(* CoDeSys 2.3 library: TcNci.lib *)
(* Libraries: TcSystem.lib*27.2.12 14:08:36, TcBaseMath.lib 27.7.04 11:07:56, TcMath.lib 23.9.04 14:15:30, tcnc.lib 10.10.08 16:55:34, standard.lib 5.6.98 11:03:02, TcBase.lib 14.5.09 11:14:08 *)

(* Global variable list: Globale_Variablen *)
VAR_GLOBAL CONSTANT

	NCI_MAX_TOOLDESC:					UDINT := 255; (* in older versions the max number of tool descriptions *)
                                               (* was restricted to 50, cf. issue 1721 & 2365*)

	NCI_MAX_READPREVIEWTABLINES	 	: UINT := 11;
	NCI_MAX_PREVIEWTABLINES 				: UINT := 20;


	(* additional TcNciItp.lib errors *)
	ErrTcNciItp_MFuncReq:			UDINT := 16#4B10;	(* m function request is missing *)
	ErrTcNciItp_ZeroShiftNo:		UDINT	:= 16#4B11;	(* zero shift number is out of range *)
	ErrTcNciItp_RParamIndex:		UDINT	:= 16#4B12;	(* index of r param or size is invalid *)
	ErrTcNciItp_DNo:					UDINT	:= 16#4B13; (* index of d number is out of range *)
	ErrTcNciItp_ItfVersion:			UDINT	:= 16#4B14; (* the cyclic channel interface does not match to the requested function/fb *)
	ErrTcNciItp_NotReady:			UDINT	:= 16#4B15;	(* not ready to support requested function *)
	ErrTcNciItp_NotEnabled:			UDINT	:= 16#4B16;	(* requested function is not enabled *)

	(* states of the interpreter *)
	NCI_INTERPRETER_INITFAILED:	UDINT	:=	0;
	NCI_INTERPRETER_IDLE:			UDINT	:=	1;
	NCI_INTERPRETER_READY:			UDINT	:=	2;
	NCI_INTERPRETER_STARTED:		UDINT	:=	3;
	NCI_INTERPRETER_SCANNING:		UDINT	:=	4;
	NCI_INTERPRETER_RUNNING:		UDINT	:=	5;
	NCI_INTERPRETER_STAY_RUNNING:	UDINT	:=	6;
	NCI_INTERPRETER_WRITETABLE:	UDINT	:=	7;
	NCI_INTERPRETER_SEARCHLINE:	UDINT	:=	8;
	NCI_INTERPRETER_END:				UDINT	:=	9;
	NCI_INTERPRETER_SINGLESTOP:	UDINT	:=	10;
	NCI_INTERPRETER_ABORTING:		UDINT	:=	11;
	NCI_INTERPRETER_ABORTED:		UDINT	:=	12;
	NCI_INTERPRETER_FAULT:			UDINT	:=	13;
	NCI_INTERPRETER_RESET:			UDINT	:=	14;
	NCI_INTERPRETER_STOP:			UDINT := 15;
	NCI_INTERPRETER_WAITFUNC:		UDINT	:=	16;
	NCI_INTERPRETER_FLUSHBUFFERS:	UDINT	:=	17;


END_VAR

VAR_GLOBAL
	g_NcPortTcNci:	UINT	:= AMSPORT_R0_NC;
END_VAR

(* Data type *)
TYPE _ST_ItpInternalPreViewTab :
STRUCT
	nDcTime 		: UDINT := 0;(* T_DCTIME32, timestamp in [ns]) from the NC-SAF(IO)-cycle related to the returned data *)
	nReserved 	: UDINT := 0;(* fill bytes (8 byte alignment) *)
	arrLines		: ARRAY[1..NCI_MAX_READPREVIEWTABLINES] OF ST_ItpPreViewTabLine;(* 272 bytes (8 + 11*24) *)
END_STRUCT
END_TYPE

(* Data type *)
TYPE E_ItpBnMode :
(
	ItpBnm_Abort	:= 0,
	ItpBnm_Adjust	:= 1,
	ItpBnm_Leave	:= 2
);
END_TYPE

(* Data type *)
TYPE E_ItpChannelType :
(
	ItpChannelTypeNone,
	ItpChannelTypeInterpreter,
	ItpChannelTypeKinematic,
	ItpChannelType_InvalidItfVer	:= 16#4B14 (* ErrTcNciItp_ItfVersion  the cyclic channel interface does not match to the requested function/fb *)
);
END_TYPE

(* Data type *)
TYPE E_ItpSingleBlockMode :
(
	ItpSingleBlockOff		:= 0,
	ItpSingleBlockNck		:= 1, (* nc-kernel single block mode *)
	ItpSingleBlockIntp	:= 16#4000 (*interpreter single block mode *)
);
END_TYPE

(* Data type *)
TYPE NciChannelFromPlc :
STRUCT
	nSkipLine		:	WORD;						(* Mask to skip lines *)
	nItpMode		:	WORD;
	nMFuncGranted	:	WORD;						(* granted signal of the M-function *)
	nReserved1		:	ARRAY[7..14] OF BYTE;
	nChaAxesOvr		:	DWORD;					(* Channel override in percent * 10000 *)
	nChaSpindleOvr	:	DWORD;
	nReserved2		:	ARRAY[23..150] OF BYTE;
END_STRUCT
END_TYPE

(* Data type *)
TYPE NciChannelToPlc :
STRUCT
	nJobNo			:	DWORD;
	nFastMFuncMask	:	ARRAY[1..5] OF DWORD;	(* Mask to evaluate fast M-functions *)
	nHskMFuncNo		:	WORD;							(* evaluate M-function with handshake *)
	nHskMFuncReq	: 	WORD;
	nHFuncValue		:	DINT;
	nSpindleRpm		:	WORD;
	nTool				:	WORD;
	nReserved1		:	ARRAY[37..132] OF BYTE; (* 37..40 nChnState *)
                                             (* 41..56 nParams *)
                                             (* 57..88 fParams *)
                                             (* 89..132 reserved *)
	nLoadedProg		:	DWORD;						(* loaded program number if exist *)
	nItpMode			:	WORD;							(* Interpreter mode *)
	nItpState		:	WORD;							(* Interpreter status *)
	nItpErrCode		:	WORD;							(* Interpreter-Channel Error Code *)
	nReserved2		:	ARRAY[143..150] OF BYTE; (*143..144 still reserved *)
                                              (*145..146 nChnId *)
                                              (*147..148 nGrpId *)
                                              (*149..150 nItfVersion *)
END_STRUCT
END_TYPE

(* Data type *)
TYPE ST_ItpEStopParams :
STRUCT
	fDec:		LREAL;
	fJerk:	LREAL;
END_STRUCT
END_TYPE

(* Data type *)
TYPE ST_ItpPreViewTab :
STRUCT
	nDcTime 		: UDINT := 0;(* T_DCTIME32, timestamp in [ns]) from the NC-SAF(IO)-cycle related to the returned data *)
	nReserved 	: UDINT := 0;(* fill bytes (8 byte alignment) *)
	arrLines		: ARRAY[1..NCI_MAX_READPREVIEWTABLINES] OF ST_ItpPreViewTabLine;(* 272 bytes (8 + 11*24) *)
END_STRUCT
END_TYPE

(* Data type *)
TYPE ST_ItpPreViewTabEx :
STRUCT
	nDcTime 		: UDINT := 0;(* T_DCTIME32, timestamp in [ns]) from the NC-SAF(IO)-cycle related to the returned data *)
	nReserved 	: UDINT := 0;(* fill bytes (8 byte alignment) *)
	arrLines		: ARRAY[1..NCI_MAX_PREVIEWTABLINES] OF ST_ItpPreViewTabLine;(* 272 bytes (8 + 11*24) *)
END_STRUCT
END_TYPE

(* Data type *)
TYPE ST_ItpPreViewTabLine :
STRUCT
	fLength 		: LREAL	:= 0.0;
	nBlockNo 	: UDINT 	:= 0;
	nHParam		: UDINT 	:= 0;
	nEntryID		: DINT 	:= 0;
	nReserved	: UDINT 	:= 0;(* fill bytes (8 byte alignment) *)
END_STRUCT
END_TYPE

(* Data type *)
TYPE ST_ItpRetrace :
STRUCT
	nReserved:	ARRAY[1..2] OF DWORD;
	fReserved:	ARRAY[1..8] OF LREAL;
END_STRUCT
END_TYPE

(* Data type *)
TYPE ToolDesc :
STRUCT
	nToolNumber:	UDINT;
	nToolType:		UDINT;
	fParam:			ARRAY[2..15] OF LREAL;
END_STRUCT
END_TYPE

(* Data type *)
TYPE ZeroShiftDesc :
STRUCT
	fShiftX:	LREAL;
	fShiftY:	LREAL;
	fShiftZ:	LREAL;
END_STRUCT
END_TYPE

(* POU MAIN, ST *)
PROGRAM MAIN
VAR
END_VAR
;
END_PROGRAM

(* POU ItpConfirmHsk, ST *)
(* Name:       ItpConfirmHsk                                *)
(* Desc:       confirms the actual m function               *)
(* Author:     kbn                                          *)
(* Date:       30-May-2001                                  *)
(* Revision:   VER 4.0.0                                    *)
(*                                                          *)
(*==========================================================*)

FUNCTION_BLOCK ItpConfirmHsk
VAR_INPUT
	bExecute:	BOOL;
END_VAR
VAR_IN_OUT
	sNciToPlc:	NciChannelToPlc;
	sPlcToNci:	NciChannelFromPlc;
END_VAR
VAR_OUTPUT
	bBusy:	BOOL	:= FALSE;
	bErr:		BOOL	:= FALSE;
	nErrId:	UDINT	:= 0;
END_VAR
VAR
	nState:		UDINT	:= 0;
END_VAR
(*
Version history:
Date          | Version    | created under      | Author          | Remark 
---------------------------------------------------------------------------------------- 
02/01/2002    | 5.1.0      | V2.8.0 (Build 719) | kbn             | modified
              |            |                    |                 | - cycle optimization
---------------------------------------------------------------------------------------- 
*) 
CASE nState OF
0:
	IF bExecute THEN
		bBusy		:= TRUE;
		bErr		:= FALSE;
		nErrId	:= 0;

		IF ItpIsHskMFunc( sNciToPlc ) THEN
			sPlcToNci.nMFuncGranted	:= 1;
			nState	:= 20;
		ELSE
			(* error - there's no request *)
			nState	:= 10;
		END_IF
	END_IF

10:
	(* error in state 0 *)
	(* to ensure a rising edge at bErr we're waiting for the next plc cycle *)
	bErr		:= TRUE;
	nErrId	:= ErrTcNciItp_MFuncReq;
	nState	:= 30;

20:
	(* wait until request bit is gone *)
	(* should be done in the next cycle *)
	IF NOT ItpIsHskMFunc( sNciToPlc ) THEN
		sPlcToNci.nMFuncGranted	:= 0;
		bBusy	:= FALSE;
		IF NOT bExecute THEN
			nState	:= 0;
		ELSE
			(* wait until bExecute has a falling edge *)
			nState	:= 30;
		END_IF
	END_IF

30:
	bBusy	:= FALSE;

	IF NOT bExecute THEN
		nState	:= 0;
	END_IF

END_CASE
END_FUNCTION_BLOCK

(* POU ItpIsHskMFunc, ST *)
(* Name:			ItpIsHskMFunc											*)
(* Desc:			determines if the handshake request bit		*)
(*					is set													*)
(* Author:	 	kbn														*)
(* Date:			30-May-2001												*)
(* Revision:	VER 4.0.0  												*)
(*==========================================================*)

FUNCTION ItpIsHskMFunc : BOOL
VAR_IN_OUT
	sNciToPlc:	NciChannelToPlc;
END_VAR
IF sNciToPlc.nHskMFuncReq <> 0 THEN
	ItpIsHskMFunc	:= TRUE;
ELSE
	ItpIsHskMFunc	:= FALSE;
END_IF
END_FUNCTION

(* POU ItpDelDtg, ST *)
(*==========================================================*)
(* ItpDelDtg																*)
(* Author:	 	kbn														*)
(* Date:			30-May-2001												*)
(* Revision:	VER 5.5.19 												*)
(* last edit:	VER 6.2.33 						                  *)
(*==========================================================*)

FUNCTION_BLOCK ItpDelDtg
VAR_INPUT
	bExecute:	BOOL;
	nChnId:		UDINT;
	tTimeOut:	TIME := DEFAULT_ADS_TIMEOUT;
END_VAR
VAR_OUTPUT
	bBusy:		BOOL	:= FALSE;
	bErr:			BOOL	:= FALSE;
	nErrId:		UDINT	:= 0;
END_VAR
VAR
	nState:		UDINT	:= 0;
	fbAdsWrite:	ADSWRITE;
END_VAR
(*
Version history:
Date          | Version    | created under      | Author          | Remark 
---------------------------------------------------------------------------------------- 
02/01/2002    | 5.1.0      | V2.8.0 (Build 719) | kbn             | modified
              |            |                    |                 | - cycle optimization
---------------------------------------------------------------------------------------- 
06/04/2002    | 5.3.8      | V2.8.0 (Build 733) | kbn             | modified
              |            |                    |                 | - cycle optimization
---------------------------------------------------------------------------------------- 
09/22/2003    | 5.4.13     | V2.9.0 (Build 947) | kbn             | adjustable target port cf. issue #2304
              |            | saved as 2.8       |                 | 
*) 
CASE nState OF

0:
	(* wait on trigger event *)
	IF bExecute THEN
		bBusy	:= TRUE;
		bErr	:= FALSE;
		nErrId	:= 0;

		fbAdsWrite(
			NETID		:= '',
			PORT		:= g_NcPortTcNci,
			IDXGRP	:= NCIDXG_CHN_FUNCS + nChnId,
			IDXOFFS	:= NCIDXO_CHNF_DELDTG,
			LEN		:= 0,
			SRCADDR	:= 0,
			WRITE		:= TRUE,
			TMOUT		:= tTimeOut);

		nState	:= 10;
	END_IF

10:
	(* execute DelDtg command *)
	fbAdsWrite();

	IF NOT fbAdsWrite.BUSY THEN
		IF NOT fbAdsWrite.ERR THEN
			IF NOT bExecute THEN
				fbAdsWrite( WRITE := FALSE );
				nState	:= 0;
			ELSE
				nState	:= 20;
			END_IF
			bBusy	:= FALSE;
		ELSE
			bErr		:= TRUE;
			nErrId	:= fbAdsWrite.ERRID;
			nState	:= 20;
		END_IF
	END_IF
20:
	fbAdsWrite( WRITE := FALSE );
	bBusy	:= FALSE;
	IF NOT bExecute THEN
		nState	:= 0;
	END_IF
END_CASE
END_FUNCTION_BLOCK

(* POU ItpDelDtgEx, ST *)
(*==========================================================*)
(* Name:			ItpDelDtgEx  											*)
(* Desc:			                                             *)
(*             trigger delete distance to go				      *)
(* Author:	 	kbn														*)
(* Date:			26-September-2006										*)
(* last edit:	VER 6.2.33 						                  *)
(*==========================================================*)
FUNCTION_BLOCK ItpDelDtgEx
VAR_IN_OUT
	sNciToPlc:	NciChannelToPlc;
END_VAR
VAR_INPUT
	bExecute:	BOOL;
	tTimeOut:	TIME := DEFAULT_ADS_TIMEOUT;
END_VAR
VAR_OUTPUT
	bBusy:		BOOL	:= FALSE;
	bErr:			BOOL	:= FALSE;
	nErrId:		UDINT	:= 0;
END_VAR
VAR
	nState:			UDINT := 0;
	fbItpDelDtg:	ItpDelDtg;
END_VAR
CASE nState OF
0:
	IF bExecute THEN
		IF ItpGetItfVersion( sNciToPlc ) > 0 THEN
			fbItpDelDtg(
				bExecute	:= TRUE,
				nChnId	:= ItpGetChannelId( sNciToPlc ),
				tTimeOut	:= tTimeOut,
				bBusy	=> bBusy,
				bErr	=> bErr,
				nErrId=> nErrId );
			nState	:= 10;
		ELSE
			bBusy		:= TRUE;
			bErr		:= TRUE;
			nErrId	:= ErrTcNciItp_ItfVersion;
			nState	:= 9999;
		END_IF
	END_IF
10:
	fbItpDelDtg();
	IF NOT fbItpDelDtg.bBusy THEN
		bBusy	:= FALSE;
		IF NOT fbItpDelDtg.bErr THEN
			IF NOT bExecute THEN
				fbItpDelDtg( bExecute := FALSE );
				nState	:= 0;
			ELSE
				nState	:= 9999;
			END_IF
		ELSE
			bErr		:= TRUE;
			nErrId	:= fbItpDelDtg.nErrId;
			nState	:= 9999;
		END_IF
	END_IF

9999:
	fbItpDelDtg( bExecute := FALSE );
	bBusy	:= FALSE;
	IF NOT bExecute THEN
		nState	:= 0;
	END_IF

END_CASE
END_FUNCTION_BLOCK

(* POU ItpGetItfVersion, ST *)
(*==========================================================*)
(* Name:			ItpGetItfVersion										*)
(* Desc:		   determines the interface version of the      *)
(*             cyclic channel interface to plc              *)
(* Author:	 	kbn														*)
(* Date:			26-September-2006										*)
(* last edit:	VER 6.1.21 cf. issue #3209                   *)
(*==========================================================*)
FUNCTION ItpGetItfVersion : UINT
VAR_INPUT
END_VAR
VAR_IN_OUT
	sNciToPlc:	NciChannelToPlc;
END_VAR
VAR
END_VAR
MEMCPY(ADR(ItpGetItfVersion), ADR(sNciToPlc.nReserved2[149]), 2);
END_FUNCTION

(* POU ItpGetChannelId, ST *)
(*==========================================================*)
(* Name:			ItpGetChannelId  										*)
(* Desc:       determines the channel id					      *)
(* Author:	 	kbn														*)
(* Date:			26-September-2006										*)
(* last edit:	VER 6.1.21 cf. issue #3209                   *)
(*==========================================================*)
FUNCTION ItpGetChannelId : UINT
VAR_INPUT
END_VAR
VAR_IN_OUT
	sNciToPlc:	NciChannelToPlc;
END_VAR
VAR
END_VAR
MEMCPY(ADR(ItpGetChannelId), ADR(sNciToPlc.nReserved2[145]), 2);
(*
IF ItpGetItfVersion( sNciToPlc ) > 0 THEN
	MEMCPY(ADR(ItpGetChannelId), ADR(sNciToPlc.nReserved2[145]), 2);
ELSE
	ItpGetChannelId	:= 0;
END_IF
*)
END_FUNCTION

(* POU ItpEnableFeederBackup, ST *)
(*==========================================================*)
(* Name:			ItpEnableFeederBackup    							*)
(* Desc:			THIS IS NOT A RELEASED IMPLEMENTATION AND    *)
(*             SUBJECT TO CHANGE                            *)
(*             enable backup feeder entries for retrace     *)
(* Author:	 	kbn														*)
(* Date:			26-november-2006										*)
(* last edit:	VER 6.2.33 						                  *)
(*==========================================================*)
FUNCTION_BLOCK ItpEnableFeederBackup
VAR_INPUT
	bEnable:		BOOL;
	bExecute:	BOOL;
	tTimeOut:	TIME := DEFAULT_ADS_TIMEOUT;
END_VAR
VAR_IN_OUT
	sNciToPlc:	NciChannelToPlc;
END_VAR
VAR_OUTPUT
	bBusy:		BOOL	:= FALSE;
	bErr:			BOOL	:= FALSE;
	nErrId:		UDINT	:= 0;
END_VAR
VAR
	nState:		UDINT	:= 0;
	nData:		UDINT	:= 0;
	fbAdsWrite:	ADSWRITE;
END_VAR
CASE nState OF
0:
	(* wait on trigger event *)
	IF bExecute THEN
		bBusy	:= TRUE;
		bErr	:= FALSE;
		nErrId	:= 0;

		IF bEnable THEN
			nData	:= 1;
		ELSE
			nData	:= 0;
		END_IF

		fbAdsWrite(
			NETID		:= '',
			PORT		:= g_NcPortTcNci,
			IDXGRP	:= NCIDXG_CHNPARMS + ItpGetChannelId(sNciToPlc:=sNciToPlc),
			IDXOFFS	:= 16#54,
			LEN		:= SIZEOF(nData),
			SRCADDR	:= ADR(nData),
			WRITE		:= TRUE,
			TMOUT		:= tTimeOut);

		nState	:= 10;
	END_IF

10:
	(* execute enable/disable feeder backup*)
	fbAdsWrite();

	IF NOT fbAdsWrite.BUSY THEN
		IF NOT fbAdsWrite.ERR THEN
			IF NOT bExecute THEN
				fbAdsWrite( WRITE := FALSE );
				nState	:= 0;
			ELSE
				nState	:= 20;
			END_IF
			bBusy	:= FALSE;
		ELSE
			bErr		:= TRUE;
			nErrId	:= fbAdsWrite.ERRID;
			nState	:= 20;
		END_IF
	END_IF
20:
	fbAdsWrite( WRITE := FALSE );
	bBusy	:= FALSE;
	IF NOT bExecute THEN
		nState	:= 0;
	END_IF
END_CASE
END_FUNCTION_BLOCK

(* POU ItpEStop, ST *)
(* Name:       ItpEStop                                     *)
(* Desc:       trigger EStop                                *)
(* Author:     kbn                                          *)
(* Date:       29-May-2002                                  *)
(* Revision:   VER 5.4.6                                    *)
(* last edit:	VER 6.2.33 						                  *)
(*==========================================================*)

FUNCTION_BLOCK ItpEStop
VAR_INPUT
	bExecute:	BOOL;
	nGrpId:		UDINT;
	fDec:			LREAL;
	fJerk:		LREAL;
	tTimeOut:	TIME := DEFAULT_ADS_TIMEOUT;
END_VAR
VAR_OUTPUT
	bBusy:	BOOL	:= FALSE;
	bErr:		BOOL	:= FALSE;
	nErrId:	UDINT	:= 0;
END_VAR
VAR
	nState:			UDINT := 0;
	fbAdsWrite:		ADSWRITE;
	stEStopParams:	ST_ItpEStopParams;
END_VAR

(*
Version history:
09/22/2003    | 5.4.13     | V2.9.0 (Build 947) | kbn             | adjustable target port cf. issue #2304
              |            | saved as 2.8       |                 |
*)
CASE nState OF
0:
	IF bExecute THEN
		bBusy		:= TRUE;
		bErr		:= FALSE;
		nErrId	:= 0;

		stEStopParams.fDec	:= fDec;
		stEStopParams.fJerk	:= fJerk;

		fbAdsWrite(
			NETID		:= '',
			PORT		:= AMSPORT_R0_NCSAF,
			IDXGRP	:= 16#3200 + nGrpId,
			IDXOFFS	:= 16#4,
			LEN		:= SIZEOF( stEStopParams ),
			SRCADDR	:= ADR( stEStopParams ),
			WRITE		:= TRUE,
			TMOUT		:= tTimeOut, );

		nState	:= 10;
	END_IF

10:
	fbAdsWrite();

	IF NOT fbAdsWrite.BUSY THEN
		IF NOT fbAdsWrite.ERR THEN
			IF NOT bExecute THEN
				fbAdsWrite( WRITE:= FALSE );
				nState	:= 0;
			ELSE
				nState	:= 20;
			END_IF
			bBusy		:= FALSE;
		ELSE
			bErr		:= TRUE;
			nErrId	:= fbAdsWrite.ERRID;
			nState	:= 20;
		END_IF
	END_IF

20:
	fbAdsWrite( WRITE:= FALSE );
	bBusy		:= FALSE;
	IF NOT bExecute THEN
		nState	:= 0;
	END_IF

END_CASE
END_FUNCTION_BLOCK

(* POU ItpEStopEx, ST *)
(*==========================================================*)
(* Name:			ItpEStopEx  											*)
(* Desc:			triggers E-Stop									   *)
(* Author:	 	kbn														*)
(* Date:			26-September-2006										*)
(* last edit:	VER 6.2.33 						                  *)
(*==========================================================*)

FUNCTION_BLOCK ItpEStopEx
VAR_IN_OUT
	sNciToPlc:	NciChannelToPlc;
END_VAR
VAR_INPUT
	bExecute:	BOOL;
	fDec:			LREAL;
	fJerk:		LREAL;
	tTimeOut:	TIME := DEFAULT_ADS_TIMEOUT;
END_VAR
VAR_OUTPUT
	bBusy:	BOOL	:= FALSE;
	bErr:		BOOL	:= FALSE;
	nErrId:	UDINT	:= 0;
END_VAR
VAR
	nState:			UDINT := 0;
	fbEStop:	ItpEStop;
END_VAR
CASE nState OF
0:
	IF bExecute THEN
		IF ItpGetItfVersion( sNciToPlc ) > 0 THEN
			fbEStop(
				bExecute	:= TRUE,
				nGrpId	:= ItpGetGroupId( sNciToPlc ),
				fDec		:= fDec,
				fJerk		:= fJerk,
				tTimeOut	:= tTimeOut,
				bBusy	=> bBusy,
				bErr	=> bErr,
				nErrId=> nErrId );
			nState	:= 10;
		ELSE
			bBusy		:= TRUE;
			bErr		:= TRUE;
			nErrId	:= ErrTcNciItp_ItfVersion;
			nState	:= 9999;
		END_IF
	END_IF
10:
	fbEStop();
	IF NOT fbEStop.bBusy THEN
		bBusy	:= FALSE;
		IF NOT fbEStop.bErr THEN
			IF NOT bExecute THEN
				fbEStop( bExecute := FALSE );
				nState	:= 0;
			ELSE
				nState	:= 9999;
			END_IF
		ELSE
			bErr		:= TRUE;
			nErrId	:= fbEStop.nErrId;
			nState	:= 9999;
		END_IF
	END_IF

9999:
	fbEStop( bExecute := FALSE );
	bBusy	:= FALSE;
	IF NOT bExecute THEN
		nState	:= 0;
	END_IF

END_CASE
END_FUNCTION_BLOCK

(* POU ItpGetGroupId, ST *)
(*==========================================================*)
(* Name:			ItpGetGroupId 											*)
(* Desc:	      determines the group id						      *)
(* Author:	 	kbn														*)
(* Date:			26-September-2006										*)
(* last edit:	VER 6.1.21 cf. issue #3209                   *)
(*==========================================================*)
FUNCTION ItpGetGroupId : UINT
VAR_INPUT
END_VAR
VAR_IN_OUT
	sNciToPlc:	NciChannelToPlc;
END_VAR
VAR
END_VAR
MEMCPY(ADR(ItpGetGroupId), ADR(sNciToPlc.nReserved2[147]), 2);
(*
IF ItpGetItfVersion( sNciToPlc ) > 0 THEN
	MEMCPY(ADR(ItpGetGroupId), ADR(sNciToPlc.nReserved2[147]), 2);
ELSE
	ItpGetGroupId	:= 0;
END_IF
*)
END_FUNCTION

(* POU ItpGetBlockNumber, ST *)
(* Name:			ItpGetBlockNumber										*)
(* Desc:			Returns the currrent block number				*)
(*						of the NC program									*)
(*	Author:	 	bw															*)
(* Date:			27-Nov-2012												*)
(* Revision:	VER 1.0.0  												*)
(*==========================================================*)
FUNCTION ItpGetBlockNumber : UDINT
VAR_IN_OUT
	sNciToPlc:	NciChannelToPlc;
END_VAR
ItpGetBlockNumber := sNciToPlc.nJobNo;
END_FUNCTION

(* POU ItpGetBottleNeckLookAhead, ST *)
(* Name:			ItpGetBottleNeckLookAhead  						*)
(* Desc:			gets the size of the look ahead for the 		*)
(*             contour collision detection (bottle neck)    *)
(* Author:	 	kbn														*)
(* Date:			26-March-2002											*)
(* Revision:	VER 5.3.4  												*)
(* last edit:	VER 6.2.33 						                  *)
(*==========================================================*)

FUNCTION_BLOCK ItpGetBottleNeckLookAhead
VAR_INPUT
	bExecute:	BOOL;
	nChnId:		UDINT;
	tTimeOut:	TIME := DEFAULT_ADS_TIMEOUT;
END_VAR
VAR_OUTPUT
	bBusy:	BOOL;
	bErr:		BOOL;
	nErrId:	UDINT;
	nLookAhead:	UDINT;
END_VAR
VAR
	nState:		UDINT	:= 0;
	fbAdsRead:	ADSREAD;
END_VAR
VAR CONSTANT
	IDXO_CHNP_BNLOOKAHEAD:	UDINT	:= 16#51;
END_VAR

(*
Version history:
09/22/2003    | 5.4.13     | V2.9.0 (Build 947) | kbn             | adjustable target port cf. issue #2304
              |            | saved as 2.8       |                 |
*)
CASE nState OF

0:
	(* wait on trigger event *)
	IF bExecute THEN
		bBusy		:= TRUE;
		bErr		:= FALSE;
		nErrId	:= 0;

		fbAdsRead(
			NETID		:= '',
			PORT		:= g_NcPortTcNci,
			IDXGRP	:= NCIDXG_CHN_PARMS + nChnId,
			IDXOFFS	:= IDXO_CHNP_BNLOOKAHEAD,
			LEN		:= SIZEOF( nLookAhead ),
			DESTADDR	:= ADR( nLookAhead ),
			READ		:= TRUE,
			TMOUT		:= tTimeOut );

		nState	:= 10;
	END_IF

10:
	fbAdsRead();

	IF NOT fbAdsRead.BUSY THEN
		IF NOT fbAdsRead.ERR THEN
			IF NOT bExecute THEN
				fbAdsRead( READ := FALSE );
				nState	:= 0;
			ELSE
				nState	:= 20;
			END_IF
			bBusy	:= FALSE;
		ELSE
			bErr		:= TRUE;
			nErrId	:= fbAdsRead.ERRID;
			nState	:= 20;
		END_IF
	END_IF

20:
	fbAdsRead( READ := FALSE );
	bBusy	:= FALSE;

	IF NOT bExecute THEN
		nState	:= 0;
	END_IF

END_CASE
END_FUNCTION_BLOCK

(* POU ItpGetBottleNeckLookAheadEx, ST *)
(*==========================================================*)
(* Name:			ItpGetBottleNeckLookAheadEx						*)
(* Desc:			gets the size of the look ahead for the 		*)
(*             contour collision detection (bottle neck)    *)
(* Author:	 	kbn														*)
(* Date:			26-September-2006										*)
(* last edit:	VER 6.2.33 						                  *)
(*==========================================================*)

FUNCTION_BLOCK ItpGetBottleNeckLookAheadEx
VAR_INPUT
	bExecute:	BOOL;
	tTimeOut:	TIME := DEFAULT_ADS_TIMEOUT;
END_VAR
VAR_IN_OUT
	sNciToPlc:	NciChannelToPlc;
END_VAR
VAR_OUTPUT
	bBusy:	BOOL;
	bErr:		BOOL;
	nErrId:	UDINT;
	nLookAhead:	UDINT;
END_VAR
VAR
	nState:		UDINT := 0;
	fbItpGetBottleNeckLookAhead:	ItpGetBottleNeckLookAhead;
END_VAR
CASE nState OF
0:
	IF bExecute THEN
		IF ItpGetItfVersion( sNciToPlc ) > 0 THEN
			fbItpGetBottleNeckLookAhead(
				bExecute	:= TRUE,
				nChnId	:= ItpGetChannelId( sNciToPlc ),
				tTimeOut	:= tTimeOut,
				bBusy	=> bBusy,
				bErr	=> bErr,
				nErrId=> nErrId,
				nLookAhead=>nLookAhead );
			nState	:= 10;
		ELSE
			bBusy		:= TRUE;
			bErr		:= TRUE;
			nErrId	:= ErrTcNciItp_ItfVersion;
			nState	:= 9999;
		END_IF
	END_IF
10:
	fbItpGetBottleNeckLookAhead( nLookAhead=>nLookAhead );
	IF NOT fbItpGetBottleNeckLookAhead.bBusy THEN
		bBusy	:= FALSE;
		IF NOT fbItpGetBottleNeckLookAhead.bErr THEN
			IF NOT bExecute THEN
				fbItpGetBottleNeckLookAhead( bExecute := FALSE, nLookAhead=>nLookAhead );
				nState	:= 0;
			ELSE
				nState	:= 9999;
			END_IF
		ELSE
			bErr		:= TRUE;
			nErrId	:= fbItpGetBottleNeckLookAhead.nErrId;
			nState	:= 9999;
		END_IF
	END_IF

9999:
	fbItpGetBottleNeckLookAhead( bExecute:=FALSE, nLookAhead=>nLookAhead );
	bBusy	:= FALSE;
	IF NOT bExecute THEN
		nState	:= 0;
	END_IF

END_CASE
END_FUNCTION_BLOCK

(* POU ItpGetBottleNeckMode, ST *)
(* Name:			ItpGetBottleNeckMode        						*)
(* Desc:			get the reaction mode for the contour        *)
(*             collision detection                          *)
(* Author:	 	kbn														*)
(* Date:			26-March-2002											*)
(* Revision:	VER 5.3.4  												*)
(* last edit:	VER 6.2.33 						                  *)
(*==========================================================*)

FUNCTION_BLOCK ItpGetBottleNeckMode
VAR_INPUT
	bExecute:			BOOL;
	nChnId:				UDINT;
	tTimeOut:			TIME := DEFAULT_ADS_TIMEOUT;
END_VAR
VAR_OUTPUT
	bBusy:	BOOL;
	bErr:		BOOL;
	nErrId:	UDINT;
	eBottleNeckMode:	E_ItpBnMode;
END_VAR
VAR
	nState:		UDINT	:= 0;
	fbAdsRead:	ADSREAD;
	nTemp:		UDINT;
END_VAR
VAR CONSTANT
	IDXO_CHNP_BNMODE:	UDINT	:= 16#50;
END_VAR

(*
Version history:
09/22/2003    | 5.4.13     | V2.9.0 (Build 947) | kbn             | adjustable target port cf. issue #2304
              |            | saved as 2.8       |                 |
*)
CASE nState OF

0:
	(* wait on trigger event *)
	IF bExecute THEN
		bBusy		:= TRUE;
		bErr		:= FALSE;
		nErrId	:= 0;

		fbAdsRead(
			NETID		:= '',
			PORT		:= g_NcPortTcNci,
			IDXGRP	:= NCIDXG_CHN_PARMS + nChnId,
			IDXOFFS	:= IDXO_CHNP_BNMODE,
			LEN		:= SIZEOF( nTemp ),
			DESTADDR	:= ADR( nTemp ),
			READ		:= TRUE,
			TMOUT		:= tTimeOut );

		nState	:= 10;
	END_IF

10:
	fbAdsRead();

	IF NOT fbAdsRead.BUSY THEN
		IF NOT fbAdsRead.ERR THEN
			eBottleNeckMode	:= UDINT_TO_INT( nTemp );
			IF NOT bExecute THEN
				fbAdsRead( READ := FALSE );
				nState	:= 0;
			ELSE
				nState	:= 20;
			END_IF
			bBusy	:= FALSE;
		ELSE
			bErr		:= TRUE;
			nErrId	:= fbAdsRead.ERRID;
			nState	:= 20;
		END_IF
	END_IF

20:
	fbAdsRead( READ := FALSE );
	bBusy	:= FALSE;

	IF NOT bExecute THEN
		nState	:= 0;
	END_IF

END_CASE
END_FUNCTION_BLOCK

(* POU ItpGetBottleNeckModeEx, ST *)
(*==========================================================*)
(* Name:			ItpGetBottleNeckModeEx								*)
(* Desc:			returns the reaction mode for the contour    *)
(*             collision detection                          *)
(* Author:	 	kbn														*)
(* Date:			26-September-2006										*)
(* last edit:	VER 6.2.33 						                  *)
(*==========================================================*)
FUNCTION_BLOCK ItpGetBottleNeckModeEx
VAR_INPUT
	bExecute:			BOOL;
	tTimeOut:			TIME := DEFAULT_ADS_TIMEOUT;
END_VAR
VAR_IN_OUT
	sNciToPlc:	NciChannelToPlc;
END_VAR
VAR_OUTPUT
	bBusy:	BOOL;
	bErr:		BOOL;
	nErrId:	UDINT;
	eBottleNeckMode:	E_ItpBnMode;
END_VAR
VAR
	nState:		UDINT := 0;
	fbItpGetBottleNeckMode:	ItpGetBottleNeckMode;
END_VAR
CASE nState OF
0:
	IF bExecute THEN
		IF ItpGetItfVersion( sNciToPlc ) > 0 THEN
			fbItpGetBottleNeckMode(
				bExecute	:= TRUE,
				nChnId	:= ItpGetChannelId( sNciToPlc ),
				tTimeOut	:= tTimeOut,
				bBusy	=> bBusy,
				bErr	=> bErr,
				nErrId=> nErrId,
				eBottleNeckMode=> eBottleNeckMode );
			nState	:= 10;
		ELSE
			bBusy		:= TRUE;
			bErr		:= TRUE;
			nErrId	:= ErrTcNciItp_ItfVersion;
			nState	:= 9999;
		END_IF
	END_IF
10:
	fbItpGetBottleNeckMode( eBottleNeckMode=>eBottleNeckMode );
	IF NOT fbItpGetBottleNeckMode.bBusy THEN
		bBusy	:= FALSE;
		IF NOT fbItpGetBottleNeckMode.bErr THEN
			IF NOT bExecute THEN
				fbItpGetBottleNeckMode( bExecute := FALSE, eBottleNeckMode=>eBottleNeckMode );
				nState	:= 0;
			ELSE
				nState	:= 9999;
			END_IF
		ELSE
			bErr		:= TRUE;
			nErrId	:= fbItpGetBottleNeckMode.nErrId;
			nState	:= 9999;
		END_IF
	END_IF

9999:
	fbItpGetBottleNeckMode( bExecute:=FALSE, eBottleNeckMode=>eBottleNeckMode );
	bBusy	:= FALSE;
	IF NOT bExecute THEN
		nState	:= 0;
	END_IF

END_CASE
END_FUNCTION_BLOCK

(* POU ItpGetChannelType, ST *)
(* Name:			ItpGetChannelType										*)
(* Desc:			Returns the Channel type as an Enum				*)
(*	Author:	 	bw															*)
(* Date:			27-Nov-2012												*)
(* Revision:	VER 1.0.0  												*)
(*==========================================================*)
FUNCTION ItpGetChannelType : E_ItpChannelType
VAR_IN_OUT
	sNciToPlc:	NciChannelToPlc;
END_VAR
IF ItpGetItfVersion(sNciToPlc)>=6 THEN
	CASE (sNciToPlc.nReserved1[37] AND 2#00000011) OF
		0:	ItpGetChannelType := ItpChannelTypeNone;
		1:	ItpGetChannelType := ItpChannelTypeInterpreter;
		2:	ItpGetChannelType := ItpChannelTypeKinematic;
		3:	ItpGetChannelType := ItpChannelTypeNone;
		ELSE
			ItpGetChannelType := ItpChannelTypeNone;
	END_CASE
ELSE
	ItpGetChannelType := ItpChannelType_InvalidItfVer;
END_IF
END_FUNCTION

(* POU ItpGetCyclicLRealOffsets, ST *)
(*==========================================================*)
(* Name:			ItpGetCyclicLRealOffsets							*)
(* Desc:			THIS IS NOT A RELEASED IMPLEMENTATION AND    *)
(*             SUBJECT TO CHANGE                            *)
(*             specifies index offsets for cylcic channel   *)
(*             interface                                    *)
(* Author:	 	kbn														*)
(* Date:			08-October-2007										*)
(* last edit:	VER 6.2.33 						                  *)
(*==========================================================*)
FUNCTION_BLOCK ItpGetCyclicLRealOffsets
VAR_INPUT
	bExecute:	BOOL;
	tTimeOut:	TIME := DEFAULT_ADS_TIMEOUT;
END_VAR
VAR_IN_OUT
	sNciToPlc:	NciChannelToPlc;
END_VAR
VAR_OUTPUT
	bBusy:		BOOL	:= FALSE;
	bErr:			BOOL	:= FALSE;
	nErrId:		UDINT	:= 0;
	nIndexOffsetParam1:	UDINT := 0;
	nIndexOffsetParam2:	UDINT := 0;
	nIndexOffsetParam3:	UDINT := 0;
	nIndexOffsetParam4:	UDINT := 0;
END_VAR
VAR
	nState:	UDINT	:= 0;
	nIndexOffsets: ARRAY[1..4] OF UDINT;
	fbAdsRead:		ADSREAD;
END_VAR
CASE nState OF
0:
	IF  bExecute THEN
		bBusy	:= TRUE;
		bErr	:= FALSE;
		nErrId	:= 0;
		fbAdsRead(
			NETID		:= '',
			PORT		:= g_NcPortTcNci,
			IDXGRP	:= NCIDXG_CHNPARMS + ItpGetChannelId(sNciToPlc:=sNciToPlc),
			IDXOFFS	:= 16#56,
			LEN		:= SIZEOF( nIndexOffsets ),
			DESTADDR	:= ADR( nIndexOffsets ),
			READ		:= TRUE,
			TMOUT		:= tTimeOut );
		nState	:= 10;
	END_IF

10:
	fbAdsRead();

	IF NOT fbAdsRead.BUSY THEN
		IF NOT fbAdsRead.ERR THEN

		nIndexOffsetParam1	:= nIndexOffsets[1] ;
		nIndexOffsetParam2	:= nIndexOffsets[2] ;
		nIndexOffsetParam3	:= nIndexOffsets[3] ;
		nIndexOffsetParam4	:= nIndexOffsets[4] ;

			IF NOT bExecute THEN
				fbAdsRead( READ := FALSE );
				nState	:= 0;
			ELSE
				nState	:= 20;
			END_IF
			bBusy		:= FALSE;
		ELSE
			bErr		:= TRUE;
			nErrId	:= fbAdsRead.ERRID;
			nState	:= 20;
		END_IF
	END_IF

20:
	fbAdsRead( READ:= FALSE );
	bBusy		:= FALSE;
	IF NOT bExecute THEN
		nState	:= 0;
	END_IF

END_CASE
END_FUNCTION_BLOCK

(* POU ItpGetCyclicUdintOffsets, ST *)
(*==========================================================*)
(* Name:			ItpGetCyclicUdintOffsets							*)
(* Desc:			THIS IS NOT A RELEASED IMPLEMENTATION AND    *)
(*             SUBJECT TO CHANGE                            *)
(*             specifies index offsets for cylcic channel   *)
(*             interface                                    *)
(* Author:	 	kbn														*)
(* Date:			08-October-2007										*)
(* last edit:	VER 6.2.33 						                  *)
(*==========================================================*)
FUNCTION_BLOCK ItpGetCyclicUdintOffsets
VAR_INPUT
	bExecute:	BOOL;
	tTimeOut:	TIME := DEFAULT_ADS_TIMEOUT;
END_VAR
VAR_IN_OUT
	sNciToPlc:	NciChannelToPlc;
END_VAR
VAR_OUTPUT
	bBusy:		BOOL	:= FALSE;
	bErr:			BOOL	:= FALSE;
	nErrId:		UDINT	:= 0;
	nIndexOffsetParam1:	UDINT := 0;
	nIndexOffsetParam2:	UDINT := 0;
	nIndexOffsetParam3:	UDINT := 0;
	nIndexOffsetParam4:	UDINT := 0;
END_VAR
VAR
	nState:	UDINT	:= 0;
	nIndexOffsets: ARRAY[1..4] OF UDINT;
	fbAdsRead:		ADSREAD;
END_VAR
CASE nState OF
0:
	IF  bExecute THEN
		bBusy	:= TRUE;
		bErr	:= FALSE;
		nErrId	:= 0;
		fbAdsRead(
			NETID		:= '',
			PORT		:= g_NcPortTcNci,
			IDXGRP	:= NCIDXG_CHNPARMS + ItpGetChannelId(sNciToPlc:=sNciToPlc),
			IDXOFFS	:= 16#55,
			LEN		:= SIZEOF( nIndexOffsets ),
			DESTADDR	:= ADR( nIndexOffsets ),
			READ		:= TRUE,
			TMOUT		:= tTimeOut );
		nState	:= 10;
	END_IF

10:
	fbAdsRead();

	IF NOT fbAdsRead.BUSY THEN
		IF NOT fbAdsRead.ERR THEN

		nIndexOffsetParam1	:= nIndexOffsets[1] ;
		nIndexOffsetParam2	:= nIndexOffsets[2] ;
		nIndexOffsetParam3	:= nIndexOffsets[3] ;
		nIndexOffsetParam4	:= nIndexOffsets[4] ;

			IF NOT bExecute THEN
				fbAdsRead( READ := FALSE );
				nState	:= 0;
			ELSE
				nState	:= 20;
			END_IF
			bBusy		:= FALSE;
		ELSE
			bErr		:= TRUE;
			nErrId	:= fbAdsRead.ERRID;
			nState	:= 20;
		END_IF
	END_IF

20:
	fbAdsRead( READ:= FALSE );
	bBusy		:= FALSE;
	IF NOT bExecute THEN
		nState	:= 0;
	END_IF

END_CASE
END_FUNCTION_BLOCK

(* POU ItpGetError, ST *)
(* Name:			ItpGetError												*)
(* Desc:			returns the error number							*)
(* Author:	 	kbn														*)
(* Date:			30-May-2001												*)
(* Revision:	VER 4.0.0  												*)
(*==========================================================*)

FUNCTION ItpGetError : UINT
VAR_IN_OUT
	sNciToPlc:	NciChannelToPlc;
END_VAR
VAR
END_VAR
ItpGetError	:= sNciToPlc.nItpErrCode;
END_FUNCTION

(* POU ItpGetGeoInfoAndHParam, ST *)
FUNCTION_BLOCK ItpGetGeoInfoAndHParam
VAR_IN_OUT
	sNciToPlc:	NciChannelToPlc;
END_VAR
VAR_OUTPUT
	stTab		: ST_ItpPreViewTab;
	nErrId	: UDINT;
END_VAR
{library private}
VAR
	fbCall	: FW_CallGenericFb := ( funGrp := GENERIC_FB_GRP_NC, funNum:= GENERIC_FB_NC_GETGEOINFOANDHPARAM );
	in 		: ARRAY[0..1] OF UDINT;(* 8 byte = nGrpId, nSubIdx *)
END_VAR
IF ItpGetItfVersion( sNciToPlc ) < 5 THEN
	nErrId	:= ErrTcNciItp_ItfVersion;
	RETURN;
END_IF


(* prepare input params *)
in[0] := ItpGetGroupId( sNciToPlc );
in[1] := 0; (* reserved for certain bit mask *)

(* call firmware function block *)
fbCall(	pWrite := ADR( in ), cbWrite:= SIZEOF( in ), pRead := ADR( stTab ), cbRead := SIZEOF( stTab ), nErrID=>nErrID );
END_FUNCTION_BLOCK

(* POU ItpGetGeoInfoAndHParamEx, ST *)
FUNCTION_BLOCK ItpGetGeoInfoAndHParamEx
(* Extended FB for reading geometric information from Nci channel 						*)
(* The H-Parameter Value is based an segment end and 10 past path values are stored		*)
VAR_IN_OUT
	sNciToPlc				: NciChannelToPlc;
END_VAR
VAR_OUTPUT
	stTab					: ST_ItpPreViewTabEx;
	nErrId 					: UDINT;
END_VAR		
{library private}
VAR
	fbCall					: FW_CallGenericFb := ( funGrp := GENERIC_FB_GRP_NC, funNum:= GENERIC_FB_NC_GETGEOINFOANDHPARAM );
	in 						: ARRAY[0..1] OF UDINT;(* 8 byte = nGrpId, nSubIdx *)

	PathInfoOffset				: DINT;
	stReadTab				: ST_ItpPreViewTab;
	stLastReadTab			: ST_ItpPreViewTab;
	stInternalTab				: ST_ItpPreViewTabEx;
	stLastInternalTab			: ST_ItpPreViewTabEx;

	NoOfNewPastEntries		: DINT;
	PathLengthCorrection		: LREAL;

	i,j						: DINT;

	DataError				: BOOL;

	(* Debug *)
	debugcounterZeroData	: UDINT;

	LastPathId				: UDINT;
END_VAR
IF ItpGetItfVersion( sNciToPlc ) < 5 THEN
	nErrId	:= ErrTcNciItp_ItfVersion;
	RETURN;
END_IF

(* prepare input params *)
in[0] := ItpGetGroupId(sNciToPlc);
in[1] := 0; (* reserved for certain bit mask *)

(* call firmware function block *)
fbCall(	pWrite := ADR( in ), cbWrite:= SIZEOF( in ), pRead := ADR( stReadTab ), cbRead := SIZEOF( stReadTab ), nErrID=>nErrId );

IF nErrId <> 0 THEN
	MEMSET(ADR(stReadTab),0,SIZEOF(stReadTab));
	MEMSET(ADR(stLastReadTab),0,SIZEOF(stLastReadTab));
	MEMSET(ADR(stInternalTab),0,SIZEOF(stInternalTab));
	MEMSET(ADR(stLastInternalTab),0,SIZEOF(stLastInternalTab));
	PathLengthCorrection := 0;
	RETURN;
END_IF

(*Init Path Position Info*)
PathInfoOffset := NCI_MAX_PREVIEWTABLINES - NCI_MAX_READPREVIEWTABLINES + 1;

FOR i := 1 TO NCI_MAX_PREVIEWTABLINES DO
	stInternalTab.arrLines[i].nEntryID:=0;
	stInternalTab.arrLines[i].nHParam:=0;
	stInternalTab.arrLines[i].fLength:=0;
	stInternalTab.arrLines[i].nBlockNo:=0;

	stTab:=stInternalTab;
END_FOR

(*Zero data recieved *)
DataError := TRUE;
FOR i := 1 TO NCI_MAX_READPREVIEWTABLINES DO
	IF  (stReadTab.arrLines[i].nEntryID > 0) THEN
		DataError := FALSE;
	END_IF
END_FOR

IF DataError THEN 
	nErrId := 9998;

	MEMSET(ADR(stReadTab),0,SIZEOF(stReadTab));
	MEMSET(ADR(stLastReadTab),0,SIZEOF(stLastReadTab));
	MEMSET(ADR(stInternalTab),0,SIZEOF(stInternalTab));
	MEMSET(ADR(stLastInternalTab),0,SIZEOF(stLastInternalTab));
	PathLengthCorrection := 0;
	debugcounterZeroData := debugcounterZeroData + 1;

	RETURN;
ELSIF nErrId = 0 THEN
	stInternalTab.nDcTime := stReadTab.nDcTime;
	stInternalTab.nReserved := stReadTab.nReserved;

	(* Create new  entries *)
	FOR i := 1 TO NCI_MAX_READPREVIEWTABLINES-1 DO
		IF stReadTab.arrLines[i+1].nEntryID > 0 THEN
			stInternalTab.arrLines[i+PathInfoOffset] := stReadTab.arrLines[i];
			stInternalTab.arrLines[i+PathInfoOffset].nHParam := stReadTab.arrLines[i+1].nHParam;
		END_IF
	END_FOR

	(* Delete buffered entries which have recieved new path lengths and calculate pathlength correction *)
	FOR i := NCI_MAX_PREVIEWTABLINES TO PathInfoOffset+1 BY -1 DO
		FOR j := NCI_MAX_PREVIEWTABLINES TO 1 BY -1 DO
			IF stLastInternalTab.arrLines[j].nEntryID = stInternalTab.arrLines[i].nEntryID THEN
				IF j > PathInfoOffset THEN
					PathLengthCorrection := stLastInternalTab.arrLines[j].fLength - stInternalTab.arrLines[i].fLength;
				END_IF
				stLastInternalTab.arrLines[j].fLength:=0;
				stLastInternalTab.arrLines[j].nEntryID:=0;
				stLastInternalTab.arrLines[j].nHParam:=0;	
			END_IF 
		END_FOR
	END_FOR

	(* Update past entries already buffered *)
	FOR i := PathInfoOffset  TO 1 BY -1 DO
		stInternalTab.arrLines[i] := stLastInternalTab.arrLines[i];
		IF stLastInternalTab.arrLines[i].nEntryID > 0 THEN
			stInternalTab.arrLines[i].fLength := stInternalTab.arrLines[i].fLength - PathLengthCorrection;
		END_IF
	END_FOR

	(*Remove Zero Enties *)
	FOR i := PathInfoOffset  TO 1 BY -1 DO
		IF stInternalTab.arrLines[i].nEntryID = 0 THEN
			IF i > 1 THEN
				FOR j := i  TO 2 BY -1 DO
					stInternalTab.arrLines[j] :=stInternalTab.arrLines[j-1]; 
				END_FOR			
			END_IF
			stLastInternalTab.arrLines[1].fLength:=0;
			stLastInternalTab.arrLines[1].nEntryID:=0;
			stLastInternalTab.arrLines[1].nHParam:=0;	
		END_IF
	END_FOR

	(* Check new past entries *)
	NoOfNewPastEntries := 0;
	FOR i := NCI_MAX_PREVIEWTABLINES TO PathInfoOffset+1 BY -1 DO
		IF stLastInternalTab.arrLines[i].nEntryID > 0 THEN
			NoOfNewPastEntries := NoOfNewPastEntries + 1;
		END_IF
	END_FOR

	(* Add new entries to FIFO, If full oldest entries are deleted *)
	IF NoOfNewPastEntries > 0 THEN
		FOR i := 1 TO (PathInfoOffset - NoOfNewPastEntries)DO
			stInternalTab.arrLines[i] := stInternalTab.arrLines[i+NoOfNewPastEntries];
		END_FOR
		j:=PathInfoOffset+1;
		FOR i := NCI_MAX_PREVIEWTABLINES TO PathInfoOffset+1 BY -1 DO
			IF stLastInternalTab.arrLines[i].nEntryID > 0 THEN
				j:=j-1;
				stInternalTab.arrLines[j] := stLastInternalTab.arrLines[i];
				stInternalTab.arrLines[j].fLength := stInternalTab.arrLines[j].fLength - PathLengthCorrection;
			END_IF
		END_FOR
	END_IF

	stTab := stInternalTab;

	stLastReadTab := stReadTab;
	stLastInternalTab := stTab;

	LastPathId := stTab.arrLines[10].nEntryID;
END_IF
END_FUNCTION_BLOCK

(* POU ItpGetGroupAxisIds, ST *)
(* Name:			ItpGetGroupAxisIds									*)
(* Desc:			Outputs a list of the Group Axes 				*)
(*						or returns an interface version error		*)
(*	Author:	 	bw															*)
(* Date:			02-Feb-2012												*)
(* Revision:	VER 1.0.0  												*)
(*==========================================================*)

FUNCTION ItpGetGroupAxisIds : DWORD
VAR_INPUT
END_VAR
VAR_IN_OUT
	nNciAxisIds 	: 	ARRAY[1..8] OF DWORD;		(*A list of Axes built in the Group*)
	sNciToPlc		:	NciChannelToPlc;
END_VAR
VAR
END_VAR
IF ItpGetItfVersion(sNciToPlc)>=6 THEN
	ItpGetGroupAxisIds	:= 0;
	nNciAxisIds[1] := BYTE_TO_DWORD(sNciToPlc.nReserved1[89]);
	nNciAxisIds[2] := BYTE_TO_DWORD(sNciToPlc.nReserved1[90]);
	nNciAxisIds[3] := BYTE_TO_DWORD(sNciToPlc.nReserved1[91]);
	nNciAxisIds[4] := BYTE_TO_DWORD(sNciToPlc.nReserved1[92]);
	nNciAxisIds[5] := BYTE_TO_DWORD(sNciToPlc.nReserved1[93]);
	nNciAxisIds[6] := BYTE_TO_DWORD(sNciToPlc.nReserved1[94]);
	nNciAxisIds[7] := BYTE_TO_DWORD(sNciToPlc.nReserved1[95]);
	nNciAxisIds[8] := BYTE_TO_DWORD(sNciToPlc.nReserved1[96]);
ELSE
	ItpGetGroupAxisIds := ErrTcNciItp_ItfVersion;
	nNciAxisIds[1] := 0;
	nNciAxisIds[2] := 0;
	nNciAxisIds[3] := 0;
	nNciAxisIds[4] := 0;
	nNciAxisIds[5] := 0;
	nNciAxisIds[6] := 0;
	nNciAxisIds[7] := 0;
	nNciAxisIds[8] := 0;
END_IF
END_FUNCTION

(* POU ItpGetHParam, ST *)
(*==========================================================*)
(* Name:			ItpGetHParam											*)
(* Desc:			determines H value from the cyclic channel	*)
(*					interface												*)
(* Author:	 	kbn														*)
(* Date:			30-May-2001												*)
(* Revision:	VER 4.0.0  												*)
(*==========================================================*)

FUNCTION ItpGetHParam : DINT
VAR_IN_OUT
	sNciToPlc:	NciChannelToPlc;
END_VAR
ItpGetHParam	:= sNciToPlc.nHFuncValue;
END_FUNCTION

(* POU ItpGetHskMFunc, ST *)
(* Name:			ItpGetHskMFunc											*)
(* Desc:			returns the number of the m function			*)
(* Author:	 	kbn														*)
(* Date:			30-May-2001												*)
(* Revision:	VER 4.0.0  												*)
(*==========================================================*)

FUNCTION ItpGetHskMFunc : INT
VAR_INPUT
	sNciToPlc:	NciChannelToPlc;
END_VAR
ItpGetHskMFunc	:= sNciToPlc.nHskMFuncNo;
END_FUNCTION

(* POU ItpGetOverridePercent, ST *)
(* Name:			ItpGetOverridePercent								*)
(* Desc:			returns the axes override in percent			*)
(* Author:	 	kbn														*)
(* Date:			30-May-2001												*)
(* Revision:	VER 4.0.0  												*)
(*==========================================================*)

FUNCTION ItpGetOverridePercent : LREAL
VAR_INPUT
	sPlcToNci:	NciChannelFromPlc;
END_VAR
ItpGetOverridePercent	:= DWORD_TO_LREAL(sPlcToNci.nChaAxesOvr) / 10000.0;
END_FUNCTION

(* POU ItpGetSParam, ST *)
(*==========================================================*)
(* Name:			ItpGetSParam											*)
(* Desc:			determines S value from the cyclic channel	*)
(*					interface												*)
(* Author:	 	kbn														*)
(* Date:			30-May-2001												*)
(* Revision:	VER 4.0.0  												*)
(*==========================================================*)

FUNCTION ItpGetSParam : UINT
VAR_IN_OUT
	sNciToPlc:	NciChannelToPlc;
END_VAR
ItpGetSParam	:= sNciToPlc.nSpindleRpm;
END_FUNCTION

(* POU ItpGetStateInterpreter, ST *)
(* Name:			ItpGetStateInterpreter								*)
(* Desc:			reads the interpreter status						*)
(* Author:	 	kbn														*)
(* Date:			15-Nov-2001												*)
(* Revision:	VER 4.1.0  												*)
(*==========================================================*)

FUNCTION ItpGetStateInterpreter : UDINT
VAR_INPUT
END_VAR
VAR_IN_OUT
	sNciToPlc:	NciChannelToPlc;
END_VAR
VAR
END_VAR
ItpGetStateInterpreter	:= sNciToPlc.nItpState;
END_FUNCTION

(* POU ItpGetTParam, ST *)
(* Name:			ItpGetTParam											*)
(* Desc:			determines T value from the cyclic channel	*)
(*					interface												*)
(* Author:	 	kbn														*)
(* Date:			30-May-2001												*)
(* Revision:	VER 4.0.0  												*)
(*==========================================================*)

FUNCTION ItpGetTParam : UINT
VAR_IN_OUT
	sNciToPlc:	NciChannelToPlc;
END_VAR
ItpGetTParam	:= sNciToPlc.nTool;
END_FUNCTION

(* POU ItpGetVersion, ST *)
FUNCTION ItpGetVersion : STRING(20)

(* Version history:
Date          | Version    | created under      | Author          | Remark 

---------------------------------------------------------------------------------------- 
2012-01-04    | 6.2.33     | V2.11  				| bw		         | Default ADS timeout added
---------------------------------------------------------------------------------------- 
2012-11-27    | 6.2.32     | V2.11  				| bw		         | New functions ItpGetChannelType and ItpGetBlockNumber
---------------------------------------------------------------------------------------- 
2012-07-25    | 6.2.31     | V2.11  				| bw		         | #9206 ItpEStop, ItpEStopEx, ItpStepOnAfterEStop and ItpStepOnAfterEStopEx improvement
---------------------------------------------------------------------------------------- 
2012-06-04    | 6.2.30     | V2.11  (Build 2223)| FAp kbn         | New fb: ItpGetGeoInfoAndHParamEx
---------------------------------------------------------------------------------------- 
2012-02-02    | 6.1.29     | V2.11	(Build 2216)| bw					| New function: ItpGetGroupAxisIds
---------------------------------------------------------------------------------------- 
2011-08-24    | 6.1.28     | V2.10.0(Build 2034)| ChristophC/kbn  | New fb: ItpGetGeoInfoAndHParam
              |            | saved as 2.11      |                 | 
---------------------------------------------------------------------------------------- 
2008-10-22    | 6.1.27     | V2.10.0(Build 1328)| kbn             | reorganisation of fb's
              |            | saved as 2.8       |                 | 
---------------------------------------------------------------------------------------- 
2008-02-22    | 6.1.26     | V2.10.0(Build 1321)| kbn             | implementation of ItpSingleStep
              |            | saved as 2.8       |                 | #3403
---------------------------------------------------------------------------------------- 
2007-10-08    | 6.1.25     | V2.10.0(Build 1319)| kbn             | beta implementation of fbs for configurable channel interface
              |            | saved as 2.8       |                 | #3373
---------------------------------------------------------------------------------------- 
2006-07-12    | 6.1.24     | V2.10.0(Build 1307)| kbn             | beta implementation of fbs for retrace
              |            | saved as 2.8       |                 | #1318
---------------------------------------------------------------------------------------- 
2006-11-08    | 6.1.23     | V2.10.0(Build 1305)| kbn             | beta implementation of fbs for retrace
              |            | saved as 2.8       |                 | #1318
---------------------------------------------------------------------------------------- 
2006-09-25    | 6.1.22     | V2.10.0(Build 1303)| kbn             | beta implementation of fb with cyclic channel interface
              |            | saved as 2.8       |                 | #3209
---------------------------------------------------------------------------------------- 
2006-06-29    | 5.5.21     | V2.10.0(Build 1301)| kbn             | changes in fb: ItpLoadProg
              |            | saved as 2.8       |                 | string length > 80 characters	#3134
---------------------------------------------------------------------------------------- 
2005-11-15    | 5.5.20     | V2.10.0(Build 1244)| kbn             | new fb: ItpResetEx
              |            | saved as 2.8       |                 | #3013
---------------------------------------------------------------------------------------- 
2005-10-18    | 5.5.19     | V2.10.0(Build 1242)| kbn             | new fb: ItpResetFastMFunc
              |            | saved as 2.8       |                 | #2996
---------------------------------------------------------------------------------------- 
2005-06-17    | 5.5.18     | V2.10.0(Build 1030)| kbn             | new fbs: 
              |            | saved as 2.8       |                 | - ItpSetZeroShiftNull
              |            |                    |                 | - ItpSetToolDescNull
              |            |                    |                 | #2900
---------------------------------------------------------------------------------------- 
2004-06-24    | 5.4.17     | V2.9.0 (Build 959) | kbn             | new fb: ItpSetSubroutinePath
              |            | saved as 2.8       |                 | #2578
---------------------------------------------------------------------------------------- 
2003-12-23    | 5.4.16     | V2.9.0 (Build 952) | kbn             | number of tool parameters #2365
              |            | saved as 2.8       |                 | 
---------------------------------------------------------------------------------------- 
2003-12-10    | 5.4.15     | V2.9.0 (Build 951) | kbn             | ItpIsEStp #2280
              |            | saved as 2.8       |                 | 
---------------------------------------------------------------------------------------- 
2003-12-10    | 5.4.14     | V2.9.0 (Build 951) | kbn             | Interpreter states cf. issue #2357
              |            | saved as 2.8       |                 | 
---------------------------------------------------------------------------------------- 
2003-09-22    | 5.4.13     | V2.9.0 (Build 947) | kbn             | adjustable target port cf. issue #2304
              |            | saved as 2.8       |                 | 
---------------------------------------------------------------------------------------- 
2003-09-22    | 5.4.12     | V2.9.0 (Build 947) | kbn             | fb's to generate a part program are moved
              |            | saved as 2.8       |                 | new TcNciUtility.lib
---------------------------------------------------------------------------------------- 
2002-11-04    | 5.4.11     | V2.9.0 (Build 906) | kbn             | cf. issue #1956
              |            |                    |                 | beta implementation & subject ot change of
              |            |                    |                 | fb's to generate a part program (teach-in)
---------------------------------------------------------------------------------------- 
2002-10-30    | 5.3.10     | V2.8.0 (Build 739) | ChristophC      | ItpStartStop: If fb is in busy state and bStop becomes rising edge,  the stop command is now send afterwards.
---------------------------------------------------------------------------------------- 
2002-09-24    | 5.3.9      | V2.9.0 (Build 901) | kbn             | cf. issue #1830
---------------------------------------------------------------------------------------- 
2002-06-04    | 5.3.8      | V2.8.0 (Build 733) | kbn             | cf. issue #1830
---------------------------------------------------------------------------------------- 
2002-05-29    | 5.3.7      | V2.8.0 (Build 733) | kbn             | beta implementation & subject to change of
              |            |                    |                 | - ItpEStop
              |            |                    |                 | - ItpStepOnAfterEStop
---------------------------------------------------------------------------------------- 
2002-05-13    | 5.3.5      | V2.8.0 (Build 733) | kbn             | parameter for max tool params
---------------------------------------------------------------------------------------- 
2002-03-26    | 5.3.4      | V2.8.0 (Build 722) | kbn             | new FB's
              |            |                    |                 | - ItpSetBottleNeckLookAhead
              |            |                    |                 | - ItpGetBottleNeckLookAhead
              |            |                    |                 | - ItpSetBottleNeckMode
              |            |                    |                 | - ItpGetBottleNeckMode
---------------------------------------------------------------------------------------- 
2002-02-28    | 5.2.3      | V2.8.0 (Build 721) | kbn             | modified
              |            |                    |                 | - start/stop priorities
---------------------------------------------------------------------------------------- 
2002-02-01    | 5.1.0      | V2.8.0 (Build 719) | kbn             | modified
              |            |                    |                 | - cycle optimization
---------------------------------------------------------------------------------------- 
2001-11-19    | 5.0.0      | V2.8.0 (Build 707) | kbn             | created
              |            |                    |                 | - based on TcNciItp.lib
---------------------------------------------------------------------------------------- 
*) 
ItpGetVersion	:= '6.002.033';
END_FUNCTION

(* POU ItpGoAhead, ST *)
(*==========================================================*)
(* Name:			ItpGoAhead												*)
(* Desc:			triggers interpreter									*)
(*					only to use in combination with @717			*)
(* Author:	 	kbn														*)
(* Date:			30-May-2001												*)
(* Revision:	VER 4.0.0  												*)
(* last edit:	VER 6.2.33 						                  *)
(*==========================================================*)

FUNCTION_BLOCK ItpGoAhead
VAR_INPUT
	bExecute:	BOOL;
	nChnId:		UDINT;
	tTimeOut:	TIME := DEFAULT_ADS_TIMEOUT;
END_VAR
VAR_OUTPUT
	bBusy:		BOOL	:= FALSE;
	bErr:			BOOL	:= FALSE;
	nErrId:		UDINT	:= 0;
END_VAR
VAR
	nState:		UDINT	:= 0;
	fbAdsWrite:	ADSWRITE;
END_VAR

(*
Version history:
Date          | Version    | created under      | Author          | Remark 
---------------------------------------------------------------------------------------- 
02/01/2002    | 5.1.0      | V2.8.0 (Build 719) | kbn             | modified
              |            |                    |                 | - cycle optimization
---------------------------------------------------------------------------------------- 
09/22/2003    | 5.4.13     | V2.9.0 (Build 947) | kbn             | adjustable target port cf. issue #2304
              |            | saved as 2.8       |                 |
*) 
CASE nState OF
0:
	(* wait on trigger event *)
	IF bExecute THEN
		bBusy	:= TRUE;
		bErr	:= FALSE;
		nErrId	:= 0;

		fbAdsWrite(
			NETID		:= '',
			PORT		:= g_NcPortTcNci,
			IDXGRP	:= NCIDXG_CHN_FUNCS + nChnId,
			IDXOFFS	:= NCIDXO_CHNF_GOAHEAD,
			LEN		:= 0,
			SRCADDR	:= 0,
			WRITE		:= TRUE,
			TMOUT		:= tTimeOut);

		nState	:= 10;
	END_IF

10:
	(* execute GoAhead command *)
	(* bugfix by kbn 02/01/2002 *)
	fbAdsWrite();
	IF NOT fbAdsWrite.BUSY THEN
		IF NOT fbAdsWrite.ERR THEN
			IF NOT bExecute THEN
				fbAdsWrite( WRITE := FALSE );
				nState	:= 0;
			ELSE
				nState	:= 20;
			END_IF
			bBusy	:= FALSE;
		ELSE
			bErr		:= TRUE;
			nErrId	:= fbAdsWrite.ERRID;
			nState	:= 20;
		END_IF
	END_IF
20:
	fbAdsWrite( WRITE := FALSE );
	bBusy	:= FALSE;
	IF NOT bExecute THEN
		nState	:= 0;
	END_IF
END_CASE
END_FUNCTION_BLOCK

(* POU ItpGoAheadEx, ST *)
(*==========================================================*)
(* Name:			ItpGoAheadEx  											*)
(* Desc:		   triggers goahead command					      *)
(* Author:	 	kbn														*)
(* Date:			26-September-2006										*)
(* last edit:	VER 6.2.33 						                  *)
(*==========================================================*)
FUNCTION_BLOCK ItpGoAheadEx
VAR_IN_OUT
	sNciToPlc:	NciChannelToPlc;
END_VAR
VAR_INPUT
	bExecute:	BOOL;
	tTimeOut:	TIME := DEFAULT_ADS_TIMEOUT;
END_VAR
VAR_OUTPUT
	bBusy:		BOOL	:= FALSE;
	bErr:			BOOL	:= FALSE;
	nErrId:		UDINT	:= 0;
END_VAR
VAR
	nState:		UDINT := 0;
	fbGoAhead:	ItpGoAhead;
END_VAR
CASE nState OF
0:
	IF bExecute THEN
		IF ItpGetItfVersion( sNciToPlc ) > 0 THEN
			fbGoAhead(
				bExecute	:= TRUE,
				nChnId	:= ItpGetChannelId( sNciToPlc ),
				tTimeOut	:= tTimeOut,
				bBusy	=> bBusy,
				bErr	=> bErr,
				nErrId=> nErrId);
			nState	:= 10;
		ELSE
			bBusy		:= TRUE;
			bErr		:= TRUE;
			nErrId	:= ErrTcNciItp_ItfVersion;
			nState	:= 9999;
		END_IF
	END_IF
10:
	fbGoAhead();
	IF NOT fbGoAhead.bBusy THEN
		bBusy	:= FALSE;
		IF NOT fbGoAhead.bErr THEN
			IF NOT bExecute THEN
				fbGoAhead( bExecute := FALSE );
				nState	:= 0;
			ELSE
				nState	:= 9999;
			END_IF
		ELSE
			bErr		:= TRUE;
			nErrId	:= fbGoAhead.nErrId;
			nState	:= 9999;
		END_IF
	END_IF

9999:
	fbGoAhead( bExecute := FALSE );
	bBusy	:= FALSE;
	IF NOT bExecute THEN
		nState	:= 0;
	END_IF

END_CASE
END_FUNCTION_BLOCK

(* POU ItpHasError, ST *)
(* Name:			ItpHasError												*)
(* Desc:			determines if the interpreter is in error		*)
(* Author:	 	kbn														*)
(* Date:			30-May-2001												*)
(* Revision:	VER 4.0.0  												*)
(*==========================================================*)

FUNCTION ItpHasError : BOOL
VAR_IN_OUT
	sNciToPlc:	NciChannelToPlc;
END_VAR
IF sNciToPlc.nItpErrCode <> 0 THEN
	ItpHasError	:= TRUE;
ELSE
	ItpHasError	:= FALSE;
END_IF
END_FUNCTION

(* POU ItpIsEStop, ST *)
(* Name:       ItpIsEStop                                   *)
(* Desc:       check if an estop is triggered               *)
(*             there is no information, if the axes already *)
(*             stand still                                  *)
(*                                                          *)
(* Author:     kbn                                          *)
(* Date:       10-Dec-2003                                  *)
(* Revision:   VER 5.4.15                                   *)
(* last edit:	VER 6.2.33 						                  *)
(*==========================================================*)
FUNCTION_BLOCK ItpIsEStop
VAR_INPUT
	bExecute:	BOOL;
	nGrpId:		UDINT;
	tTimeOut:	TIME := DEFAULT_ADS_TIMEOUT;
END_VAR
VAR_OUTPUT
	bBusy:	BOOL	:= FALSE;
	bEStop:	BOOL	:= FALSE;
	bErr:		BOOL	:= FALSE;
	nErrId:	UDINT	:= 0;
END_VAR
VAR
	nState:			UDINT := 0;
	nReadParam:		UINT	:= 0;
	fbAdsRead:		ADSREAD;
END_VAR
CASE nState OF

0:
	IF bExecute THEN
		bBusy		:= TRUE;
		bErr		:= FALSE;
		nErrId	:= 0;

		fbAdsRead(
			NETID		:= '',
			PORT		:= g_NcPortTcNci,
			IDXGRP	:= 16#3100 + nGrpId,
			IDXOFFS	:= 16#11,
			LEN		:= SIZEOF( nReadParam ),
			DESTADDR	:= ADR( nReadParam ),
			READ		:= TRUE,
			TMOUT		:= tTimeOut );

		nState	:= 10;
	END_IF

10:
	fbAdsRead();

	IF NOT fbAdsRead.BUSY THEN

		IF nReadParam = 0 THEN
			bEStop	:= FALSE;
		ELSE
			bEStop	:= TRUE;
		END_IF

		IF NOT fbAdsRead.ERR THEN
			IF NOT bExecute THEN
				fbAdsRead( READ := FALSE );
				nState	:= 0;
			ELSE
				nState	:= 20;
			END_IF
			bBusy	:= FALSE;
		ELSE
			bErr		:= TRUE;
			nErrId	:= fbAdsRead.ERRID;
			nState	:= 20;
		END_IF
	END_IF

20:
	fbAdsRead( Read := FALSE );
	bBusy	:= FALSE;
	IF NOT bExecute THEN
		nState	:= 0;
	END_IF
END_CASE
END_FUNCTION_BLOCK

(* POU ItpIsEStopEx, ST *)
(*==========================================================*)
(* Name:			ItpIsEStopEx             							*)
(* Desc:			THIS IS NOT A RELEASED IMPLEMENTATION AND    *)
(*             SUBJECT TO CHANGE                            *)
(*					it requires at least interface version 2     *)
(*             (GetItfVersion)                              *)
(*             checks if an estop is active or requested    *)
(*             there is no information about if the axis    *)
(*             already stands still                         *)
(* Author:	 	kbn														*)
(* Date:			26-november-2006										*)
(* last edit:	VER 6.1.23 cf. issue #1318                   *)
(*==========================================================*)
FUNCTION ItpIsEStopEx : BOOL
VAR_INPUT
END_VAR
VAR_IN_OUT
	sNciToPlc:	NciChannelToPlc;
END_VAR
VAR
	nChnStateDWord:	DWORD;
END_VAR
IF ItpGetItfVersion( sNciToPlc ) < 2 THEN
	ItpIsEStopEx	:= FALSE;
ELSE
	MEMCPY(ADR(nChnStateDWord), ADR(sNciToPlc.nReserved1[37]), SIZEOF(nChnStateDWord));
	IF nChnStateDWord.8 THEN
		ItpIsEStopEx	:= TRUE;
	ELSE
		ItpIsEStopEx	:= FALSE;
	END_IF
END_IF
END_FUNCTION

(* POU ItpIsFastMFunc, ST *)
(* Name:			ItpIsFastMFunc											*)
(* Desc:			determines if the fast m-func bit of the		*)
(*					specified function is set							*)
(* Author:	 	kbn														*)
(* Date:			30-May-2001												*)
(* Revision:	VER 4.0.0  												*)
(*==========================================================*)

FUNCTION ItpIsFastMFunc : BOOL
VAR_INPUT
	nFastMFuncNo:	INT;
END_VAR
VAR_IN_OUT
	sNciToPlc:	NciChannelToPlc;
END_VAR
VAR CONSTANT
	nMFuncMin:	INT	:= 0;
	nMFuncMax:	INT	:= 159;
END_VAR
VAR
	nArrayPos:	INT	:= 0;
	nBitPos:		SINT	:= 0;
END_VAR
IF nFastMFuncNo < nMFuncMin OR nFastMFuncNo > nMFuncMax THEN
	(* this is not a valid m function number, so return false *)
	ItpIsFastMFunc	:= FALSE;
ELSE
	(* ok - valid range *)

	(* determine fast m func word number *)
	nArrayPos	:= nFastMFuncNo / 32 + 1;	(* array is one based *)
	nBitPos		:= INT_TO_SINT( nFastMFuncNo MOD 32 );
	ItpIsFastMFunc	:= GETBIT32( sNciToPlc.nFastMFuncMask[nArrayPos], nBitPos);
END_IF
END_FUNCTION

(* POU ItpIsFeederBackupEnabled, ST *)
(*==========================================================*)
(* Name:			ItpIsFeederBackupEnabled  							*)
(* Desc:			THIS IS NOT A RELEASED IMPLEMENTATION AND    *)
(*             SUBJECT TO CHANGE                            *)
(*             is feeder backup for retrace enabled?        *)
(* Author:	 	kbn														*)
(* Date:			07-december-2006										*)
(* last edit:	VER 6.2.33 						                  *)
(*==========================================================*)
FUNCTION_BLOCK ItpIsFeederBackupEnabled
VAR_INPUT
	bExecute:	BOOL;
	tTimeOut:	TIME := DEFAULT_ADS_TIMEOUT;
END_VAR
VAR_IN_OUT
	sNciToPlc:	NciChannelToPlc;
END_VAR
VAR_OUTPUT
	bBusy:		BOOL	:= FALSE;
	bEnabled:	BOOL	:= FALSE;
	bErr:			BOOL	:= FALSE;
	nErrId:		UDINT	:= 0;
END_VAR
VAR
	nState:		UDINT	:= 0;
	nData:		UDINT	:= 0;
	fbAdsRead:	ADSREAD;
END_VAR
CASE nState OF
0:
	(* wait on trigger event *)
	IF bExecute THEN
		bBusy	:= TRUE;
		bErr	:= FALSE;
		nErrId	:= 0;

		fbAdsRead(
			NETID		:= '',
			PORT		:= g_NcPortTcNci,
			IDXGRP	:= NCIDXG_CHNPARMS + ItpGetChannelId(sNciToPlc:=sNciToPlc),
			IDXOFFS	:= 16#54,
			LEN		:= SIZEOF(nData),
			DESTADDR	:= ADR(nData),
			READ		:= TRUE,
			TMOUT		:= tTimeOut );

		nState	:= 10;
	END_IF

10:
	fbAdsRead();

	IF NOT fbAdsRead.BUSY THEN
		IF NOT fbAdsRead.ERR THEN
			IF nData.0 THEN
				bEnabled	:= TRUE;
			ELSE
				bEnabled	:= FALSE;
			END_IF
			IF NOT bExecute THEN
				fbAdsRead( READ := FALSE );
				nState	:= 0;
			ELSE
				nState	:= 20;
			END_IF
			bBusy	:= FALSE;
		ELSE
			bErr		:= TRUE;
			nErrId	:= fbAdsRead.ERRID;
			nState	:= 20;
		END_IF
	END_IF
20:
	fbAdsRead( READ := FALSE );
	bBusy	:= FALSE;
	IF NOT bExecute THEN
		nState	:= 0;
	END_IF
END_CASE
END_FUNCTION_BLOCK

(* POU ItpIsFeedFromBackupList, ST *)
(*==========================================================*)
(* Name:			ItpIsFeedFromBackupList   							*)
(* Desc:			THIS IS NOT A RELEASED IMPLEMENTATION AND    *)
(*             SUBJECT TO CHANGE                            *)
(*             checks if the actual executed feeder entry   *)
(*             is from backup list                          *)
(* Author:	 	kbn														*)
(* Date:			26-november-2006										*)
(* last edit:	VER 6.1.23 cf. issue #1318                   *)
(*==========================================================*)
FUNCTION ItpIsFeedFromBackupList : BOOL
VAR_INPUT
END_VAR
VAR_IN_OUT
	sNciToPlc:	NciChannelToPlc;
END_VAR
VAR
	nChnStateDWord:	DWORD;
END_VAR
IF ItpGetItfVersion( sNciToPlc ) < 3 THEN
	ItpIsFeedFromBackupList	:= FALSE;
ELSE
	MEMCPY(ADR(nChnStateDWord), ADR(sNciToPlc.nReserved1[37]), SIZEOF(nChnStateDWord));
	IF nChnStateDWord.10 THEN
		ItpIsFeedFromBackupList	:= TRUE;
	ELSE
		ItpIsFeedFromBackupList	:= FALSE;
	END_IF
END_IF
END_FUNCTION

(* POU ItpLoadProg, FBD *)
FUNCTION_BLOCK ItpLoadProg
VAR_INPUT
	bExecute	:	BOOL;
	nChnId		:	UDINT;
	sPrg		:	STRING(255);
	nLength		:	UDINT;
	tTimeOut		:	TIME := DEFAULT_ADS_TIMEOUT;
END_VAR
VAR_OUTPUT
	bBusy		:	BOOL;
	bErr			:	BOOL;
	nErrId		:	UDINT;
END_VAR
VAR CONSTANT
	(* NC ADS Index Offsets for CHANNEL Functions *)
	NCIDXO_CHNF_LOADPROGNAME			: UDINT := 16#00000004;
END_VAR
VAR
	AdsWrite1	:	ADSWRITE;

END_VAR
(*
Version history:
09/22/2003    | 5.4.13     | V2.9.0 (Build 947) | kbn             | adjustable target port cf. issue #2304
              |            | saved as 2.8       |                 |
-----------------------------------------------------------------------------------------------------------------
06/29/2006    | 5.5.21     | V2.10.0(Build 1301)| kbn             | changes in fb: ItpLoadProg
              |            | saved as 2.8       |                 | string length > 80 characters	#3134

*)
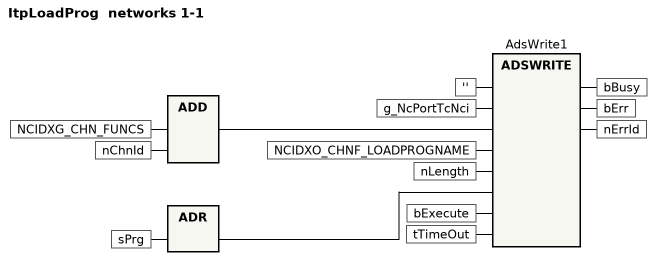
_FBD_ (* Function Block Diagram *)
NETWORK 1
	AdsWrite1:ADSWRITE('', g_NcPortTcNci, ADD(NCIDXG_CHN_FUNCS, nChnId), NCIDXO_CHNF_LOADPROGNAME, nLength, ADR(sPrg), bExecute, tTimeOut, out 2 => bErr, out 3 => nErrId) => bBusy
_END_FBD_
END_FUNCTION_BLOCK

(* POU ItpLoadProgEx, ST *)
(*==========================================================*)
(* Name:			ItpLoadProgEx 											*)
(* Desc:	      loads nc program								      *)
(* Author:	 	kbn														*)
(* Date:			26-September-2006										*)
(* last edit:	VER 6.2.33 						                  *)
(*==========================================================*)
FUNCTION_BLOCK ItpLoadProgEx
VAR_IN_OUT
	sNciToPlc:	NciChannelToPlc;
END_VAR
VAR_INPUT
	bExecute	:	BOOL;
	sPrg		:	STRING(255);
	nLength	:	UDINT;
	tTimeOut	:	TIME := DEFAULT_ADS_TIMEOUT;
END_VAR
VAR_OUTPUT
	bBusy		:	BOOL	:= FALSE;
	bErr		:	BOOL	:= FALSE;
	nErrId	:	UDINT	:= 0;
END_VAR
VAR
	nState:		UDINT := 0;
	fbLoadProg:	ItpLoadProg;
END_VAR
(*
	nChnId	:	UDINT;
*)
CASE nState OF
0:
	IF bExecute THEN
		IF ItpGetItfVersion( sNciToPlc ) > 0 THEN
			fbLoadProg(
				bExecute	:= TRUE,
				nChnId	:= ItpGetChannelId( sNciToPlc ),
				sPrg		:= sPrg,
				nLength	:= nLength,
				tTimeOut	:= tTimeOut,
				bBusy	=> bBusy,
				bErr	=> bErr,
				nErrId=> nErrId);
			nState	:= 10;
		ELSE
			bBusy		:= TRUE;
			bErr		:= TRUE;
			nErrId	:= ErrTcNciItp_ItfVersion;
			nState	:= 9999;
		END_IF
	END_IF
10:
	fbLoadProg();
	IF NOT fbLoadProg.bBusy THEN
		bBusy	:= FALSE;
		IF NOT fbLoadProg.bErr THEN
			IF NOT bExecute THEN
				fbLoadProg( bExecute := FALSE );
				nState	:= 0;
			ELSE
				nState	:= 9999;
			END_IF
		ELSE
			bErr		:= TRUE;
			nErrId	:= fbLoadProg.nErrId;
			nState	:= 9999;
		END_IF
	END_IF

9999:
	fbLoadProg( bExecute := FALSE );
	bBusy	:= FALSE;
	IF NOT bExecute THEN
		nState	:= 0;
	END_IF

END_CASE
END_FUNCTION_BLOCK

(* POU ItpReadCyclicLRealParam1, ST *)
(*==========================================================*)
(* Name:			ItpReadCyclicLRealParam1							*)
(* Desc:			THIS IS NOT A RELEASED IMPLEMENTATION AND    *)
(*             SUBJECT TO CHANGE                            *)
(*             reads an lreal value from cyclic interface   *)
(* Author:	 	kbn														*)
(* Date:			08-October-2007										*)
(* last edit:	VER 6.1.25 cf. issue #3373                   *)
(*==========================================================*)
FUNCTION ItpReadCyclicLRealParam1 : LREAL
VAR_INPUT
END_VAR
VAR_IN_OUT
	sNciToPlc:	NciChannelToPlc;
END_VAR
VAR
END_VAR
IF ItpGetItfVersion( sNciToPlc ) >= 4  THEN
	MEMCPY(ADR(ItpReadCyclicLRealParam1), ADR(sNciToPlc.nReserved1[57]), 8);
ELSE
	ItpReadCyclicLRealParam1	:= 0.0;
END_IF
END_FUNCTION

(* POU ItpReadCyclicLRealParam2, ST *)
(*==========================================================*)
(* Name:			ItpReadCyclicLRealParam2							*)
(* Desc:			THIS IS NOT A RELEASED IMPLEMENTATION AND    *)
(*             SUBJECT TO CHANGE                            *)
(*             reads an lreal value from cyclic interface   *)
(* Author:	 	kbn														*)
(* Date:			08-October-2007										*)
(* last edit:	VER 6.1.25 cf. issue #3373                   *)
(*==========================================================*)
FUNCTION ItpReadCyclicLRealParam2 : LREAL
VAR_INPUT
END_VAR
VAR_IN_OUT
	sNciToPlc:	NciChannelToPlc;
END_VAR
VAR
END_VAR
IF ItpGetItfVersion( sNciToPlc ) >= 4  THEN
	MEMCPY(ADR(ItpReadCyclicLRealParam2), ADR(sNciToPlc.nReserved1[65]), 8);
ELSE
	ItpReadCyclicLRealParam2	:= 0.0;
END_IF
END_FUNCTION

(* POU ItpReadCyclicLRealParam3, ST *)
(*==========================================================*)
(* Name:			ItpReadCyclicLRealParam3							*)
(* Desc:			THIS IS NOT A RELEASED IMPLEMENTATION AND    *)
(*             SUBJECT TO CHANGE                            *)
(*             reads an lreal value from cyclic interface   *)
(* Author:	 	kbn														*)
(* Date:			08-October-2007										*)
(* last edit:	VER 6.1.25 cf. issue #3373                   *)
(*==========================================================*)
FUNCTION ItpReadCyclicLRealParam3 : LREAL
VAR_INPUT
END_VAR
VAR_IN_OUT
	sNciToPlc:	NciChannelToPlc;
END_VAR
VAR
END_VAR
IF ItpGetItfVersion( sNciToPlc ) >= 4  THEN
	MEMCPY(ADR(ItpReadCyclicLRealParam3), ADR(sNciToPlc.nReserved1[73]), 8);
ELSE
	ItpReadCyclicLRealParam3	:= 0.0;
END_IF
END_FUNCTION

(* POU ItpReadCyclicLRealParam4, ST *)
(*==========================================================*)
(* Name:			ItpReadCyclicLRealParam3							*)
(* Desc:			THIS IS NOT A RELEASED IMPLEMENTATION AND    *)
(*             SUBJECT TO CHANGE                            *)
(*             reads an lreal value from cyclic interface   *)
(* Author:	 	kbn														*)
(* Date:			08-October-2007										*)
(* last edit:	VER 6.1.25 cf. issue #3373                   *)
(*==========================================================*)
FUNCTION ItpReadCyclicLRealParam4 : LREAL
VAR_INPUT
END_VAR
VAR_IN_OUT
	sNciToPlc:	NciChannelToPlc;
END_VAR
VAR
END_VAR
IF ItpGetItfVersion( sNciToPlc ) >= 4  THEN
	MEMCPY(ADR(ItpReadCyclicLRealParam4), ADR(sNciToPlc.nReserved1[81]), 8);
ELSE
	ItpReadCyclicLRealParam4	:= 0.0;
END_IF
END_FUNCTION

(* POU ItpReadCyclicUdintParam1, ST *)
(*==========================================================*)
(* Name:			ItpReadCyclicUdintParam1							*)
(* Desc:			THIS IS NOT A RELEASED IMPLEMENTATION AND    *)
(*             SUBJECT TO CHANGE                            *)
(*             reads an udint value from cyclic interface   *)
(* Author:	 	kbn														*)
(* Date:			08-October-2007										*)
(* last edit:	VER 6.1.25 cf. issue #3373                   *)
(*==========================================================*)
FUNCTION ItpReadCyclicUdintParam1 : UDINT
VAR_INPUT
END_VAR
VAR_IN_OUT
	sNciToPlc:	NciChannelToPlc;
END_VAR
VAR
END_VAR
IF ItpGetItfVersion( sNciToPlc ) >= 4  THEN
	MEMCPY(ADR(ItpReadCyclicUdintParam1), ADR(sNciToPlc.nReserved1[41]), 4);
ELSE
	ItpReadCyclicUdintParam1	:= 0;
END_IF
END_FUNCTION

(* POU ItpReadCyclicUdintParam2, ST *)
(*==========================================================*)
(* Name:			ItpReadCyclicUdintParam2							*)
(* Desc:			THIS IS NOT A RELEASED IMPLEMENTATION AND    *)
(*             SUBJECT TO CHANGE                            *)
(*             reads an udint value from cyclic interface   *)
(* Author:	 	kbn														*)
(* Date:			08-October-2007										*)
(* last edit:	VER 6.1.25 cf. issue #3373                   *)
(*==========================================================*)
FUNCTION ItpReadCyclicUdintParam2 : UDINT
VAR_INPUT
END_VAR
VAR_IN_OUT
	sNciToPlc:	NciChannelToPlc;
END_VAR
VAR
END_VAR
IF ItpGetItfVersion( sNciToPlc ) >= 4  THEN
	MEMCPY(ADR(ItpReadCyclicUdintParam2), ADR(sNciToPlc.nReserved1[45]), 4);
ELSE
	ItpReadCyclicUdintParam2	:= 0;
END_IF
END_FUNCTION

(* POU ItpReadCyclicUdintParam3, ST *)
(*==========================================================*)
(* Name:			ItpReadCyclicUdintParam3							*)
(* Desc:			THIS IS NOT A RELEASED IMPLEMENTATION AND    *)
(*             SUBJECT TO CHANGE                            *)
(*             reads an udint value from cyclic interface   *)
(* Author:	 	kbn														*)
(* Date:			08-October-2007										*)
(* last edit:	VER 6.1.25 cf. issue #3373                   *)
(*==========================================================*)
FUNCTION ItpReadCyclicUdintParam3 : UDINT
VAR_INPUT
END_VAR
VAR_IN_OUT
	sNciToPlc:	NciChannelToPlc;
END_VAR
VAR
END_VAR
IF ItpGetItfVersion( sNciToPlc ) >= 4  THEN
	MEMCPY(ADR(ItpReadCyclicUdintParam3), ADR(sNciToPlc.nReserved1[49]), 4);
ELSE
	ItpReadCyclicUdintParam3	:= 0;
END_IF
END_FUNCTION

(* POU ItpReadCyclicUdintParam4, ST *)
(*==========================================================*)
(* Name:			ItpReadCyclicUdintParam4							*)
(* Desc:			THIS IS NOT A RELEASED IMPLEMENTATION AND    *)
(*             SUBJECT TO CHANGE                            *)
(*             reads an udint value from cyclic interface   *)
(* Author:	 	kbn														*)
(* Date:			08-October-2007										*)
(* last edit:	VER 6.1.25 cf. issue #3373                   *)
(*==========================================================*)
FUNCTION ItpReadCyclicUdintParam4 : UDINT
VAR_INPUT
END_VAR
VAR_IN_OUT
	sNciToPlc:	NciChannelToPlc;
END_VAR
VAR
END_VAR
IF ItpGetItfVersion( sNciToPlc ) >= 4  THEN
	MEMCPY(ADR(ItpReadCyclicUdintParam4), ADR(sNciToPlc.nReserved1[53]), 4);
ELSE
	ItpReadCyclicUdintParam4	:= 0;
END_IF
END_FUNCTION

(* POU ItpReadRParams, ST *)
FUNCTION_BLOCK ItpReadRParams
VAR_INPUT
	bExecute	:	BOOL;
	nChnId		:	UDINT;
	pAddr		:	DWORD;
	nIndex		:	DINT;
	nCount		:	DINT;
	tTimeOut		:	TIME := DEFAULT_ADS_TIMEOUT;
END_VAR
VAR_OUTPUT
	bBusy:	BOOL	:= FALSE;
	bErr:		BOOL	:= FALSE;
	nErrId:	UDINT	:= 0;
END_VAR
VAR CONSTANT
	(* NC ADS Index Offsets for CHANNEL Processdata *)
	NCIDXO_CHNP_RPARAMS				: UDINT := 16#10000000;

	(* states *)
	IDLE		:	INT := 0;
	START		:	INT := 1;
	WAIT		:	INT := 2;
	ERROR		:	INT := 10;
	QUIT		:	INT := 20;
END_VAR
VAR
	Dummy		:	LREAL;
	state		:	INT := IDLE;

	(* instances *)
	AdsRead1	:	ADSREAD;
END_VAR

(*
Version history:
Date          | Version    | created under      | Author          | Remark 
---------------------------------------------------------------------------------------- 
02/01/2002    | 5.1.0      | V2.8.0 (Build 719) | kbn             | modified
              |            |                    |                 | - cycle optimization
---------------------------------------------------------------------------------------- 
09/22/2003    | 5.4.13     | V2.9.0 (Build 947) | kbn             | adjustable target port cf. issue #2304
              |            | saved as 2.8       |                 |
*) 
(* statemachine *)
CASE state OF

	IDLE:
		IF bExecute THEN
			bBusy := TRUE;
			bErr := FALSE;
			nErrId := 0;

			AdsRead1.NETID			:= '';
			AdsRead1.PORT			:= g_NcPortTcNci;
			AdsRead1.IDXGRP		:= NCIDXG_CHN_IOAREA + nChnId;
			AdsRead1.IDXOFFS		:= NCIDXO_CHNP_RPARAMS + nIndex;
			AdsRead1.LEN			:= nCount * SIZEOF(Dummy);
			AdsRead1.DESTADDR	:= pAddr;
			AdsRead1.TMOUT		:= tTimeOut;

			IF ((nIndex-1) + nCount) > 999 THEN
				nErrId := ErrTcNciItp_RParamIndex;
				state := ERROR;
			ELSE
				IF AdsRead1.READ OR AdsRead1.BUSY THEN
					AdsRead1( READ := FALSE );
				ELSE
					AdsRead1( READ := TRUE );
					state := WAIT;
				END_IF
			END_IF
		END_IF

	WAIT:
		AdsRead1();
		IF NOT AdsRead1.BUSY THEN
			IF NOT AdsRead1.ERR THEN
				IF NOT bExecute THEN
					state := IDLE;
				ELSE
					state := QUIT;
				END_IF
				bBusy := FALSE;
			ELSE
				nErrId := AdsRead1.ERRID;
				state := ERROR;
			END_IF
			AdsRead1( READ := FALSE );
		END_IF

(*
	c.f. issue 1581
		IF NOT AdsRead1.BUSY THEN
			IF NOT AdsRead1.ERR THEN
				bBusy := FALSE;
				state := QUIT;
			ELSE
				nErrId := AdsRead1.ERRID;
				state := ERROR;
			END_IF
			AdsRead1( READ := FALSE );
		END_IF
*)
	ERROR:
		bErr := TRUE;
		bBusy := FALSE;
		IF NOT bExecute THEN
			state := IDLE;
		ELSE
			state := QUIT;
		END_IF

	QUIT:
		IF NOT bExecute THEN
			state := IDLE;
		END_IF

END_CASE
END_FUNCTION_BLOCK

(* POU ItpReadRParamsEx, ST *)
(*==========================================================*)
(* Name:			ItpReadRParamsEx										*)
(* Desc:		   reads the r-parameters from a given channel  *)
(* Author:	 	kbn														*)
(* Date:			26-September-2006										*)
(* last edit:	VER 6.2.33 						                  *)
(*==========================================================*)

FUNCTION_BLOCK ItpReadRParamsEx
VAR_IN_OUT
	sNciToPlc:	NciChannelToPlc;
END_VAR
VAR_INPUT
	bExecute	:	BOOL;
	pAddr		:	DWORD;
	nIndex	:	DINT;
	nCount	:	DINT;
	tTimeOut	:	TIME := DEFAULT_ADS_TIMEOUT;
END_VAR
VAR_OUTPUT
	bBusy		:	BOOL	:= FALSE;
	bErr		:	BOOL	:= FALSE;
	nErrId	:	UDINT	:= 0;
END_VAR
VAR
	nState:		UDINT := 0;
	fbItpReadRParams:	ItpReadRParams;
END_VAR
CASE nState OF
0:
	IF bExecute THEN
		IF ItpGetItfVersion( sNciToPlc ) > 0 THEN
			fbItpReadRParams(
				bExecute	:= TRUE,
				nChnId	:= ItpGetChannelId( sNciToPlc ),
				pAddr		:= pAddr,
				nIndex	:= nIndex,
				nCount	:= nCount,
				tTimeOut	:= tTimeOut,
				bBusy	=> bBusy,
				bErr	=> bErr,
				nErrId=> nErrId );
			nState	:= 10;
		ELSE
			bBusy		:= TRUE;
			bErr		:= TRUE;
			nErrId	:= ErrTcNciItp_ItfVersion;
			nState	:= 9999;
		END_IF
	END_IF
10:
	fbItpReadRParams();
	IF NOT fbItpReadRParams.bBusy THEN
		bBusy	:= FALSE;
		IF NOT fbItpReadRParams.bErr THEN
			IF NOT bExecute THEN
				fbItpReadRParams( bExecute := FALSE );
				nState	:= 0;
			ELSE
				nState	:= 9999;
			END_IF
		ELSE
			bErr		:= TRUE;
			nErrId	:= fbItpReadRParams.nErrId;
			nState	:= 9999;
		END_IF
	END_IF

9999:
	fbItpReadRParams( bExecute := FALSE );
	bBusy	:= FALSE;
	IF NOT bExecute THEN
		nState	:= 0;
	END_IF

END_CASE
END_FUNCTION_BLOCK

(* POU ItpReadToolDesc, ST *)
(* Name:			ItpReadToolDesc										*)
(* Desc:			determines the actual tool description for 	*)
(*             the specified tool row (d word)              *)
(* Author:	 	kbn														*)
(* Date:			30-May-2001												*)
(* Revision:	VER 4.0.0  												*)
(* last edit:	VER 6.2.33 						                  *)
(*==========================================================*)

FUNCTION_BLOCK ItpReadToolDesc
VAR_INPUT
	bExecute:	BOOL;
	nChnId:		UDINT;
	nDNo:			UDINT;
	tTimeOut:	TIME := DEFAULT_ADS_TIMEOUT;
END_VAR
VAR_IN_OUT
	sToolDesc:	ToolDesc;
END_VAR
VAR_OUTPUT
	bBusy:		BOOL	:= FALSE;
	bErr:			BOOL	:= FALSE;
	nErrId:		UDINT	:= 0;
END_VAR
VAR
	nState:		UDINT	:= 0;
	nOffsetDNo:		UDINT	:= 0;
	fbReadParams:	ADSREAD;
END_VAR
VAR CONSTANT
	DNO_MIN:		UDINT	:= 1;
(*	DNO_MAX:		UDINT := 50;*)

	(* index offsets *)
	IDXOFFSET_PARAMS:	UDINT	:= 16#00040000;
END_VAR

(*
Version history:
09/22/2003    | 5.4.13     | V2.9.0 (Build 947) | kbn             | adjustable target port cf. issue #2304
              |            | saved as 2.8       |                 |
*)
CASE nState OF
0:
	IF bExecute THEN
		bBusy		:= TRUE;
		bErr		:= FALSE;
		nErrId	:= 0;

		nState	:= 10;
	END_IF

10:
	(* check nDNo *)
	IF nDNo < DNO_MIN OR nDNo > NCI_MAX_TOOLDESC THEN
		(* d number out of range *)
		bErr		:= TRUE;
		nErrId	:= ErrTcNciItp_DNo;
		nState	:= 999;
	ELSE
		nOffsetDNo	:= SHL( nDNo,  8 );
		fbReadParams(
			NETID		:= '',
			PORT		:= g_NcPortTcNci,
			IDXGRP	:= NCIDXG_CHN_PARMS + nChnId,
			IDXOFFS	:= IDXOFFSET_PARAMS + nOffsetDNo,
			LEN		:= SIZEOF( sToolDesc ),
			DESTADDR	:= ADR( sToolDesc ),
			READ		:= TRUE,
			TMOUT		:= tTimeOut);

		nState	:= 20;
	END_IF

20:
	(* wait until all read commands are executed *)
	fbReadParams();

	IF NOT fbReadParams.BUSY THEN
		IF NOT fbReadParams.ERR THEN
			nState	:= 30;
		ELSE
			bErr		:= TRUE;
			nErrId	:= fbReadParams.ERRID;
			nState	:= 999;
		END_IF
	END_IF
30:
	bBusy	:= FALSE;

	fbReadParams( READ := FALSE );

	IF NOT bExecute THEN
		nState	:= 0;
	END_IF

999:
	(* error handling *)
	bBusy	:= FALSE;

	fbReadParams( READ := FALSE );

	IF NOT bExecute THEN
		nState	:= 0;
	END_IF

END_CASE
END_FUNCTION_BLOCK

(* POU ItpReadToolDescEx, ST *)
(*==========================================================*)
(* Name:			ItpReadToolDescEx										*)
(* Desc:			determines the actual tool description for 	*)
(*             the specified tool row (d word)              *)
(* Author:	 	kbn														*)
(* Date:			26-September-2006										*)
(* last edit:	VER 6.2.33 						                  *)
(*==========================================================*)

FUNCTION_BLOCK ItpReadToolDescEx
VAR_INPUT
	bExecute:	BOOL;
	nDNo:			UDINT;
	tTimeOut:	TIME := DEFAULT_ADS_TIMEOUT;
END_VAR
VAR_IN_OUT
	sNciToPlc:	NciChannelToPlc;
	sToolDesc:	ToolDesc;
END_VAR
VAR_OUTPUT
	bBusy		:	BOOL	:= FALSE;
	bErr		:	BOOL	:= FALSE;
	nErrId	:	UDINT	:= 0;
END_VAR
VAR
	nState:		UDINT := 0;
	fbReadToolDesc:	ItpReadToolDesc;
END_VAR
CASE nState OF
0:
	IF bExecute THEN
		IF ItpGetItfVersion( sNciToPlc ) > 0 THEN
			fbReadToolDesc(
				bExecute	:= TRUE,
				nChnId	:= ItpGetChannelId( sNciToPlc ),
				nDNo		:= nDNo,
				tTimeOut	:= tTimeOut,
				sToolDesc:= sToolDesc,
				bBusy	=> bBusy,
				bErr	=> bErr,
				nErrId=> nErrId );
			nState	:= 10;
		ELSE
			bBusy		:= TRUE;
			bErr		:= TRUE;
			nErrId	:= ErrTcNciItp_ItfVersion;
			nState	:= 9999;
		END_IF
	END_IF
10:
	fbReadToolDesc( sToolDesc:=sToolDesc );
	IF NOT fbReadToolDesc.bBusy THEN
		bBusy	:= FALSE;
		IF NOT fbReadToolDesc.bErr THEN
			IF NOT bExecute THEN
				fbReadToolDesc( bExecute:=FALSE, sToolDesc:=sToolDesc );
				nState	:= 0;
			ELSE
				nState	:= 9999;
			END_IF
		ELSE
			bErr		:= TRUE;
			nErrId	:= fbReadToolDesc.nErrId;
			nState	:= 9999;
		END_IF
	END_IF

9999:
	fbReadToolDesc( bExecute:=FALSE, sToolDesc:=sToolDesc );
	bBusy	:= FALSE;
	IF NOT bExecute THEN
		nState	:= 0;
	END_IF

END_CASE
END_FUNCTION_BLOCK

(* POU ItpReadZeroShift, ST *)
(* Name:			ItpReadZeroShift										*)
(* Desc:			determines the actual zero shift	values of 	*)
(*             the specified zero shift number              *)
(* Author:	 	kbn														*)
(* Date:			30-May-2001												*)
(* Revision:	VER 4.0.0  												*)
(* last edit:	VER 6.2.33 						                  *)
(*==========================================================*)

FUNCTION_BLOCK ItpReadZeroShift
VAR_INPUT
	bExecute:	BOOL;
	nChnId:		UDINT;
	nZsNo:		UDINT;
	tTimeOut:	TIME := DEFAULT_ADS_TIMEOUT;
END_VAR
VAR_IN_OUT
	sZeroShiftDesc:	ZeroShiftDesc;
END_VAR
VAR_OUTPUT
	bBusy:		BOOL	:= FALSE;
	bErr:			BOOL	:= FALSE;
	nErrId:		UDINT	:= 0;
END_VAR
VAR
	nState:		UDINT	:= 0;
	nOffsetZsNo:	UDINT	:= 0;
	fbAdsReadX:	ADSREAD;
	fbAdsReadY:	ADSREAD;
	fbAdsReadZ:	ADSREAD;
	fShiftX:		LREAL;
	fShiftY:		LREAL;
	fShiftZ:		LREAL;
END_VAR
VAR CONSTANT
	ZSNO_MIN:		UDINT	:= 54;
	ZSNOADJ_MAX:	UDINT := 57;	(* max adjustable zero shift number *)
	ZSNO_MAX:		UDINT := 59;

	NCIDXO_CHNP_ITPZS:	UDINT	:= 16#00010000;
	ZeroShiftX:				UDINT	:= 16#00000100;
	ZeroShiftY:				UDINT	:= 16#00000200;
	ZeroShiftZ:				UDINT	:= 16#00000300;
END_VAR
(*
Version history:
09/22/2003    | 5.4.13     | V2.9.0 (Build 947) | kbn             | adjustable target port cf. issue #2304
              |            | saved as 2.8       |                 |
*)
CASE nState OF
0:
	IF bExecute THEN
		bBusy		:= TRUE;
		bErr		:= FALSE;
		nErrId	:= 0;

		nState	:= 10;
	END_IF

10:
	(* check zero shift number *)
	IF ( nZsNo < ZSNO_MIN ) OR ( nZsNo > ZSNO_MAX ) THEN
		(* error *)
		bErr		:= TRUE;
		nErrId	:= ErrTcNciItp_ZeroShiftNo;
		nState	:= 999;
	ELSE
		(* IndexOffset	0x00010K0L
							K: index of axis X=1, Y=2, Z=3
							L: zero shift number
								G54F (fine)	= 1
							 	G54G (raw) 	= 2
								G55F (fine) = 3 ...
		*)

		(* determine additional index offset for zero shift number *)
		IF nZsNo <= ZSNOADJ_MAX THEN
			nOffsetZsNo	:= (nZsNo - ZSNO_MIN)*2 + 1;
		ELSE
			nOffsetZsNo	:= nZsNo - ZSNO_MIN + 5;
		END_IF

		(* read zero shift - fine *)
		fbAdsReadX(
			NETID		:= '',
			PORT		:= g_NcPortTcNci,
			IDXGRP	:= NCIDXG_CHN_PARMS + nChnId,
			IDXOFFS	:= NCIDXO_CHNP_ITPZS + ZeroShiftX + nOffsetZsNo,
			LEN		:= SIZEOF( fShiftX ),
			DESTADDR	:= ADR( fShiftX ),
			READ		:= TRUE,
			TMOUT		:= tTimeOut );

		fbAdsReadY(
			NETID		:= '',
			PORT		:= g_NcPortTcNci,
			IDXGRP	:= NCIDXG_CHN_PARMS + nChnId,
			IDXOFFS	:= NCIDXO_CHNP_ITPZS + ZeroShiftY + nOffsetZsNo,
			LEN		:= SIZEOF( fShiftY ),
			DESTADDR	:= ADR( fShiftY ),
			READ		:= TRUE,
			TMOUT		:= tTimeOut );

		fbAdsReadZ(
			NETID		:= '',
			PORT		:= g_NcPortTcNci,
			IDXGRP	:= NCIDXG_CHN_PARMS + nChnId,
			IDXOFFS	:= NCIDXO_CHNP_ITPZS + ZeroShiftZ + nOffsetZsNo,
			LEN		:= SIZEOF( fShiftZ ),
			DESTADDR	:= ADR( fShiftZ ),
			READ		:= TRUE,
			TMOUT		:= tTimeOut );

		nState	:= 20;
	END_IF

20:
	(* wait until zero shift fine is read *)

	fbAdsReadX();
	fbAdsReadY();
	fbAdsReadZ();

	IF fbAdsReadX.ERR THEN
		bErr		:= TRUE;
		nErrId	:= fbAdsReadX.ERRID;
		nState	:= 999;
	END_IF

	IF fbAdsReadY.ERR AND NOT bERR THEN
		bERR		:= TRUE;
		nErrId	:= fbAdsReadY.ERRID;
		nState	:= 999;
	END_IF

	IF fbAdsReadZ.Err AND NOT bERR THEN
		bErr		:= TRUE;
		nErrId	:= fbAdsReadZ.ERRID;
		nState	:= 999;
	END_IF

	IF ( NOT fbAdsReadX.BUSY ) AND  ( NOT fbAdsReadY.BUSY ) AND ( NOT fbAdsReadZ.BUSY ) THEN
		IF NOT bERR THEN
			nState	:= 30;
		END_IF
	END_IF

30:
	fbAdsReadX( READ := FALSE );
	fbAdsReadY( READ := FALSE );
	fbAdsReadZ( READ := FALSE );

	sZeroShiftDesc.fShiftX	:= fShiftX;
	sZeroShiftDesc.fShiftY	:= fShiftY;
	sZeroShiftDesc.fShiftZ	:= fShiftZ;

	nState	:= 40;

40:
		(* determine additional index offset for zero shift number *)
		IF nZsNo <= ZSNOADJ_MAX THEN
			nOffsetZsNo	:= (nZsNo - ZSNO_MIN)*2 + 2;
			nState	:= 45;
		ELSE
			(* skip second read. in this case we've just one parameter *)
			fShiftX	:= 0.0;
			fShiftY	:= 0.0;
			fShiftZ	:= 0.0;

			nState	:= 60;
		END_IF

45:
	(* read zero shift - raw *)
	fbAdsReadX(
		NETID		:= '',
		PORT		:= g_NcPortTcNci,
		IDXGRP	:= NCIDXG_CHN_PARMS + nChnId,
		IDXOFFS	:= NCIDXO_CHNP_ITPZS + ZeroShiftX + (nZsNo - ZSNO_MIN)*2 + 2,
		LEN		:= SIZEOF( fShiftX ),
		DESTADDR	:= ADR( fShiftX ),
		READ		:= TRUE,
		TMOUT		:= tTimeOut );

	fbAdsReadY(
		NETID		:= '',
		PORT		:= g_NcPortTcNci,
		IDXGRP	:= NCIDXG_CHN_PARMS + nChnId,
		IDXOFFS	:= NCIDXO_CHNP_ITPZS + ZeroShiftY + (nZsNo - ZSNO_MIN)*2 + 2,
		LEN		:= SIZEOF( fShiftY ),
		DESTADDR	:= ADR( fShiftY ),
		READ		:= TRUE,
		TMOUT		:= tTimeOut );

	fbAdsReadZ(
		NETID		:= '',
		PORT		:= g_NcPortTcNci,
		IDXGRP	:= NCIDXG_CHN_PARMS + nChnId,
		IDXOFFS	:= NCIDXO_CHNP_ITPZS + ZeroShiftZ + (nZsNo - ZSNO_MIN)*2 + 2,
		LEN		:= SIZEOF( fShiftZ ),
		DESTADDR	:= ADR( fShiftZ ),
		READ		:= TRUE,
		TMOUT		:= tTimeOut );

	nState	:= 50;

50:
	(* wait until zero shift raw is read *)

	fbAdsReadX();
	fbAdsReadY();
	fbAdsReadZ();

	IF fbAdsReadX.ERR THEN
		bErr		:= TRUE;
		nErrId	:= fbAdsReadX.ERRID;
		nState	:= 999;
	END_IF

	IF fbAdsReadY.ERR AND NOT bERR THEN
		bERR		:= TRUE;
		nErrId	:= fbAdsReadY.ERRID;
		nState	:= 999;
	END_IF

	IF fbAdsReadZ.Err AND NOT bERR THEN
		bErr		:= TRUE;
		nErrId	:= fbAdsReadZ.ERRID;
		nState	:= 999;
	END_IF

	IF ( NOT fbAdsReadX.BUSY ) AND  ( NOT fbAdsReadY.BUSY ) AND ( NOT fbAdsReadZ.BUSY ) THEN
		IF NOT bERR THEN
			sZeroShiftDesc.fShiftX	:= sZeroShiftDesc.fShiftX + fShiftX;
			sZeroShiftDesc.fShiftY	:= sZeroShiftDesc.fShiftY + fShiftY;
			sZeroShiftDesc.fShiftZ	:= sZeroShiftDesc.fShiftZ + fShiftZ;

			nState	:= 60;
		END_IF
	END_IF

60:
	fbAdsReadX( READ := FALSE );
	fbAdsReadY( READ := FALSE );
	fbAdsReadZ( READ := FALSE );

	bBusy	:= FALSE;

	IF NOT bExecute THEN
		nState	:= 0;
	END_IF

999:
	(* error handling *)
	bBusy	:= FALSE;
	fbAdsReadX( READ := FALSE );
	fbAdsReadY( READ := FALSE );
	fbAdsReadZ( READ := FALSE );

	IF NOT bExecute THEN
		nState	:= 0;
	END_IF
END_CASE
END_FUNCTION_BLOCK

(* POU ItpReadZeroShiftEx, ST *)
(*==========================================================*)
(* Name:			ItpReadZeroShiftEx									*)
(* Desc:			THIS IS NOT A RELEASED IMPLEMENTATION AND    *)
(*             SUBJECT TO CHANGE                            *)
(*     			determines the actual zero shift	values of 	*)
(*             the specified zero shift number              *)
(* Author:	 	kbn														*)
(* Date:			26-September-2006										*)
(* last edit:	VER 6.2.33 						                  *)
(*==========================================================*)

FUNCTION_BLOCK ItpReadZeroShiftEx
VAR_INPUT
	bExecute:	BOOL;
	nZsNo:		UDINT;
	tTimeOut:	TIME := DEFAULT_ADS_TIMEOUT;
END_VAR
VAR_IN_OUT
	sNciToPlc:			NciChannelToPlc;
	sZeroShiftDesc:	ZeroShiftDesc;
END_VAR
VAR_OUTPUT
	bBusy:	BOOL	:= FALSE;
	bErr:		BOOL	:= FALSE;
	nErrId:	UDINT	:= 0;
END_VAR
VAR
	nState:		UDINT := 0;
	fbReadZeroShift:	ItpReadZeroShift;
END_VAR
CASE nState OF
0:
	IF bExecute THEN
		IF ItpGetItfVersion( sNciToPlc ) > 0 THEN
			fbReadZeroShift(
				bExecute	:= TRUE,
				nChnId	:= ItpGetChannelId( sNciToPlc ),
				nZsNo		:= nZsNo,
				tTimeOut	:= tTimeOut,
				sZeroShiftDesc:= sZeroShiftDesc,
				bBusy	=> bBusy,
				bErr	=> bErr,
				nErrId=> nErrId );
			nState	:= 10;
		ELSE
			bBusy		:= TRUE;
			bErr		:= TRUE;
			nErrId	:= ErrTcNciItp_ItfVersion;
			nState	:= 9999;
		END_IF
	END_IF
10:
	fbReadZeroShift( sZeroShiftDesc := sZeroShiftDesc );
	IF NOT fbReadZeroShift.bBusy THEN
		bBusy	:= FALSE;
		IF NOT fbReadZeroShift.bErr THEN
			IF NOT bExecute THEN
				fbReadZeroShift( bExecute:=FALSE, sZeroShiftDesc:=sZeroShiftDesc );
				nState	:= 0;
			ELSE
				nState	:= 9999;
			END_IF
		ELSE
			bErr		:= TRUE;
			nErrId	:= fbReadZeroShift.nErrId;
			nState	:= 9999;
		END_IF
	END_IF

9999:
	fbReadZeroShift( bExecute:=FALSE, sZeroShiftDesc:=sZeroShiftDesc );
	bBusy	:= FALSE;
	IF NOT bExecute THEN
		nState	:= 0;
	END_IF

END_CASE
END_FUNCTION_BLOCK

(* POU ItpReset, FBD *)
FUNCTION_BLOCK ItpReset
VAR_INPUT
	bExecute	:	BOOL;
	nChnId		:	UDINT;
	tTimeOut		:	TIME := DEFAULT_ADS_TIMEOUT;
END_VAR

VAR_OUTPUT
	bBusy		:	BOOL;
	bErr			:	BOOL;
	nErrId		:	UDINT;
END_VAR

VAR
	AdsWrite1	:	ADSWRITE;
	Buffer		:	BYTE := 0;
END_VAR
(*
Version history:
09/22/2003    | 5.4.13     | V2.9.0 (Build 947) | kbn             | adjustable target port cf. issue #2304
              |            | saved as 2.8       |                 |
*)
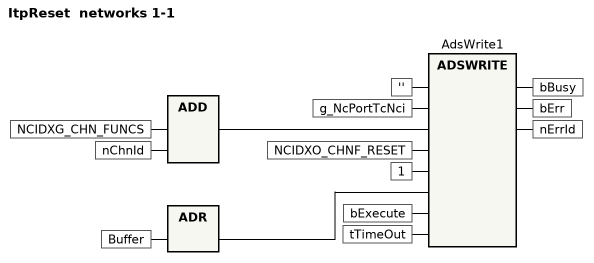
_FBD_ (* Function Block Diagram *)
NETWORK 1
	AdsWrite1:ADSWRITE('', g_NcPortTcNci, ADD(NCIDXG_CHN_FUNCS, nChnId), NCIDXO_CHNF_RESET, 1, ADR(Buffer), bExecute, tTimeOut, out 2 => bErr, out 3 => nErrId) => bBusy
_END_FBD_
END_FUNCTION_BLOCK

(* POU ItpResetEx, ST *)
(*==========================================================*)
(* Name:			ItpResetEx												*)
(* Desc:			THIS IS NOT A RELEASED IMPLEMENTAITON AND    *)
(*             SUBJECT TO CHANGE                            *)
(*             executes a stop before the reset is done     *)
(* Author:	 	kbn														*)
(* Date:			15-November-2005										*)
(* last edit:	VER 6.2.33 						                  *)
(*==========================================================*)
FUNCTION_BLOCK ItpResetEx
VAR_INPUT
	bExecute		:	BOOL;
	nGrpId		:	UDINT;
	nChnId		:	UDINT;
	tTimeOut		:	TIME := DEFAULT_ADS_TIMEOUT;
END_VAR
VAR_OUTPUT
	bBusy			:	BOOL	:= FALSE;
	bErr			:	BOOL	:= FALSE;
	nErrId		:	UDINT	:= 0;
END_VAR
VAR
	nState:	UDINT	:= 0;
	fbRTrig:R_TRIG;
	fbNciStop:ItpStartStop;
	bExecNciStop:	BOOL	:= FALSE;
	fbAdsReadActualConfig:ADSREAD;
	bExecReadActualConfig:	BOOL	:= FALSE;
	nAxisIds:	ARRAY[0..7] OF UDINT;
	nCounter:	UDINT	:= 0;
	bAllAxesStandStill:	BOOL	:= FALSE;
	fbAdsReadVelo:	ARRAY[0..7] OF ADSREAD;
	fSetVelo: ARRAY[0..7] OF LREAL;
	bExecReadVelo: ARRAY[0..7] OF BOOL	:= FALSE;
	fbGenericReset:ItpReset;
	bExecGenericReset:	BOOL	:= FALSE;
END_VAR
fbRTrig( CLK:=bExecute);
IF fbRTrig.Q THEN
	bErr	:= FALSE;
	nErrId	:= 0;
	nState	:= 0;
	bExecNciStop	:= FALSE;
	bExecReadActualConfig	:= FALSE;
	bAllAxesStandStill	:= FALSE;
	bExecGenericReset	:= FALSE;
	FOR nCounter:= 0 TO 7 DO
		bExecReadVelo[nCounter]	:= FALSE;
		fSetVelo[nCounter]	:= 0.0;
	END_FOR
END_IF

CASE nState OF
0:
	IF bExecute THEN
		bBusy	:= TRUE;
		nState	:= 10; (*goto ten to ensure that fbNciStop is called with false once *)
	END_IF

10:
	(* stop interpolation channel, at first *)
	bExecNciStop	:= TRUE;
	nState	:= 11;
11:
	IF fbNciStop.bErr THEN
		bBusy	:= FALSE;
		bErr	:= fbNciStop.bErr;
		nErrId	:= fbNciStop.nErrId;
	ELSIF NOT fbNciStop.bBusy THEN
		nState	:= 20;
	END_IF

20:
	(* wait until all axes stand still *)
	(* first read actual configuration *)
	bExecReadActualConfig	:= TRUE;
	nState	:= 21;
21:
	IF fbAdsReadActualConfig.ERR THEN
		bBusy	:= FALSE;
		bErr	:= TRUE;
		nErrId	:= fbAdsReadActualConfig.ERRID;
	ELSIF NOT fbAdsReadActualConfig.BUSY THEN
		nState	:= 22;
	END_IF
22:
	(* check if all axes stand still *)
	(* therefore check the setvelo - doing just a logical check with AxisIsNotMoving is not enough in case of override 0 *)
	FOR nCounter := 0 TO 7 DO
		IF nAxisIds[nCounter] <> 0 THEN
			bExecReadVelo[nCounter]	:= TRUE;
		END_IF
	END_FOR
	nState	:= 23;
23:
	nState	:= 24; (* will be set to 23 if one is still busy or in error *)
	FOR nCounter := 0 TO 7 DO
		IF fbAdsReadVelo[nCounter].ERR AND nAxisIds[nCounter] <> 0 THEN
			bBusy	:= FALSE;
			bErr	:= TRUE;
			nErrId	:= fbAdsReadVelo[nCounter].ERRID;
			nState	:= 23;
			EXIT;
		ELSIF fbAdsReadVelo[nCounter].BUSY THEN
			nState	:= 23;
		END_IF
	END_FOR
24:
	(* all velos are read - so check it now *)
	bAllAxesStandStill	:= TRUE;
	FOR nCounter := 0 TO 7 DO
		IF ABS(fSetVelo[nCounter]) > 0.001 THEN
			bAllAxesStandStill	:= FALSE;
		END_IF
		bExecReadVelo[nCounter]	:= FALSE;
	END_FOR
	IF NOT bAllAxesStandStill THEN
		(* read again *)
		nState	:= 22;
	ELSE
		(* all axes stand still *)
		nState	:= 30;
	END_IF

30:
	bExecGenericReset	:= TRUE;
	nState	:= 31;
31:
	IF fbGenericReset.bErr THEN
		bBusy	:= FALSE;
		bErr	:= TRUE;
		nErrId	:= fbGenericReset.nErrId;
	ELSIF NOT fbGenericReset.bBusy THEN
		nState	:= 32;
	END_IF

32:
	bBusy	:= FALSE;
	IF NOT bExecute THEN
		nState	:= 0;
	END_IF

END_CASE


fbNciStop( bStart:= FALSE, bStop:= bExecNciStop, nChnId:= nChnId, tTimeOut:= tTimeOut );
fbAdsReadActualConfig( NETID:= '', PORT:= 500, IDXGRP:= 16#3100 + nGrpId, IDXOFFS:= 16#552, LEN:= SIZEOF( nAxisIds ), DESTADDR:= ADR( nAxisIds ), READ:=bExecReadActualConfig, TMOUT:=tTimeOut);
FOR nCounter:= 0 TO 7 DO
	fbAdsReadVelo[nCounter]( NETID:= '', PORT:= 500, IDXGRP:= 16#4100 + nAxisIds[nCounter], IDXOFFS:= 16#E, LEN:= SIZEOF( fSetVelo[nCounter] ), DESTADDR:= ADR( fSetVelo[nCounter] ), READ:=bExecReadVelo[nCounter], TMOUT:=tTimeOut);
END_FOR
fbGenericReset( bExecute:= bExecGenericReset, nChnId:= nChnId, tTimeOut:= tTimeOut );
END_FUNCTION_BLOCK

(* POU ItpStartStop, ST *)
FUNCTION_BLOCK ItpStartStop
VAR_INPUT
	bStart		:	BOOL;
	bStop			:	BOOL;
	nChnId		:	UDINT;
	tTimeOut		:	TIME := DEFAULT_ADS_TIMEOUT;
END_VAR
VAR_OUTPUT
	bBusy		:	BOOL	:= FALSE;
	bErr		:	BOOL	:= FALSE;
	nErrId	:	UDINT	:= 0;
END_VAR
VAR
	fbAdsWrite		:	ADSWRITE;
	RisingStart		:	R_TRIG;
	RisingStop		:	R_TRIG;
	x_nStep 			: 	INT := 0;
	x_bStop			: 	BOOL;
END_VAR
(*
Version history:
Date          | Version    | created under      | Author          | Remark 
---------------------------------------------------------------------------------------- 
02/28/2002    | 5.2.3      | V2.8.0 (Build 721) | kbn             | modified
              |            |                    |                 | - start/stop priorities
---------------------------------------------------------------------------------------- 
10/30/2002    | 5.3.10     | V2.8.0 (Build 739 )| ChristophC      | If fb is in busy state and bStop becomes rising edge,  the stop command is now send afterwards.
---------------------------------------------------------------------------------------- 
09/22/2003    | 5.4.13     | V2.9.0 (Build 947) | kbn             | adjustable target port cf. issue #2304
              |            | saved as 2.8       |                 |
*) 
RisingStart( CLK := bStart );
RisingStop( CLK := bStop );

IF RisingStop.Q THEN
	x_bStop := TRUE;
END_IF

CASE x_nStep OF
	0:
		IF ( RisingStop.Q OR RisingStart.Q ) THEN

			IF RisingStop.Q THEN  (* STOP hat Vorrang vor START *)
				x_nStep := 10;
			ELSIF RisingStart.Q THEN
				x_nStep := 20;
			END_IF

			fbAdsWrite( WRITE := FALSE ); (*reset fb*)
			bBusy := TRUE;
			bErr := FALSE;
			nErrId := 0;
		END_IF
END_CASE

(*#########################################################################################*)
CASE x_nStep OF
	10:
		fbAdsWrite(
						NETID		:= '',
						PORT 		:= g_NcPortTcNci,
						IDXGRP	:= NCIDXG_CHN_FUNCS + nChnId,
						IDXOFFS	:= NCIDXO_CHNF_STOP,
						LEN		:= 0,
						SRCADDR	:= 0,
						WRITE		:= TRUE,
						TMOUT		:= tTimeOut );
		x_nStep := 200;
		x_bStop := FALSE;
	20:
		fbAdsWrite(
						NETID		:= '',
						PORT 		:= g_NcPortTcNci,
						IDXGRP 	:= NCIDXG_CHN_FUNCS + nChnId,
						IDXOFFS	:= NCIDXO_CHNF_STARTPROG,
						LEN		:= 0,
						SRCADDR	:= 0,
						WRITE		:= TRUE,
						TMOUT		:= tTimeOut );
		x_nStep := 200;

	200:
		fbAdsWrite( WRITE := FALSE );
		IF NOT fbAdsWrite.Busy  THEN
			IF x_bStop THEN
				fbAdsWrite( WRITE := FALSE );
				x_nStep := 10;
			ELSE
				bBusy := FALSE;
				bErr := fbAdsWrite.ERR;
				nErrId := fbAdsWrite.ERRID;
				x_nStep := 0;
			END_IF
		END_IF
END_CASE
END_FUNCTION_BLOCK

(* POU ItpResetEx2, ST *)
(*==========================================================*)
(* Name:			ItpResetEx2												*)
(* Desc:		   executes a stop before the reset is done     *)
(* Author:	 	kbn														*)
(* Date:			26-September-2006										*)
(* last edit:	VER 6.2.33 						                  *)
(*==========================================================*)

FUNCTION_BLOCK ItpResetEx2
VAR_INPUT
	bExecute		:	BOOL;
	tTimeOut		:	TIME := DEFAULT_ADS_TIMEOUT;
END_VAR
VAR_IN_OUT
	sNciToPlc:	NciChannelToPlc;
END_VAR
VAR_OUTPUT
	bBusy:	BOOL	:= FALSE;
	bErr:		BOOL	:= FALSE;
	nErrId:	UDINT	:= 0;
END_VAR
VAR
	nState:		UDINT := 0;
	fbResetEx:	ItpResetEx;
END_VAR
CASE nState OF
0:
	IF bExecute THEN
		IF ItpGetItfVersion( sNciToPlc ) > 0 THEN
			fbResetEx(
				bExecute	:= TRUE,
				nGrpId	:= ItpGetGroupId( sNciToPlc ),
				nChnId	:= ItpGetChannelId( sNciToPlc ),
				tTimeOut	:= tTimeOut,
				bBusy	=> bBusy,
				bErr	=> bErr,
				nErrId=> nErrId );
			nState	:= 10;
		ELSE
			bBusy		:= TRUE;
			bErr		:= TRUE;
			nErrId	:= ErrTcNciItp_ItfVersion;
			nState	:= 9999;
		END_IF
	END_IF
10:
	fbResetEx();
	IF NOT fbResetEx.bBusy THEN
		bBusy	:= FALSE;
		IF NOT fbResetEx.bErr THEN
			IF NOT bExecute THEN
				fbResetEx( bExecute := FALSE );
				nState	:= 0;
			ELSE
				nState	:= 9999;
			END_IF
		ELSE
			bErr		:= TRUE;
			nErrId	:= fbResetEx.nErrId;
			nState	:= 9999;
		END_IF
	END_IF

9999:
	fbResetEx( bExecute:=FALSE );
	bBusy	:= FALSE;
	IF NOT bExecute THEN
		nState	:= 0;
	END_IF

END_CASE
END_FUNCTION_BLOCK

(* POU ItpResetFastMFunc, ST *)
(*==========================================================*)
(* Name:			ItpResetFastMFunc 									*)
(* Desc:			resets specified fast m-func						*)
(* Author:	 	kbn														*)
(* Date:			18-October-2005										*)
(* Revision:	VER 5.4.19 	#2996										*)
(* last edit:	VER 6.2.33 						                  *)
(*==========================================================*)

FUNCTION_BLOCK ItpResetFastMFunc
VAR_INPUT
	bExecute:	BOOL;
	nChnId:		UDINT;
	nMFuncNo:	UINT;
	tTimeOut:	TIME := DEFAULT_ADS_TIMEOUT;
END_VAR
VAR_OUTPUT
	bBusy:	BOOL	:= FALSE;
	bErr:		BOOL	:= FALSE;
	nErrId:	UDINT	:= 0;
END_VAR
VAR
	nState:		UDINT	:= 0;
	fbAdsWrite:	ADSWRITE;
END_VAR
CASE nState OF

0:
	(* wait on trigger event *)
	IF bExecute THEN
		bBusy	:= TRUE;
		bErr	:= FALSE;
		nErrId	:= 0;

		fbAdsWrite(
			NETID		:= '',
			PORT		:= g_NcPortTcNci,
			IDXGRP	:= NCIDXG_CHN_FUNCS + nChnId,
			IDXOFFS	:= 16#60,
			LEN		:= SIZEOF(nMFuncNo),
			SRCADDR	:= ADR(nMFuncNo),
			WRITE		:= TRUE,
			TMOUT		:= tTimeOut);

		nState	:= 10;
	END_IF

10:
	(* execute AdsWrite command *)
	fbAdsWrite();

	IF NOT fbAdsWrite.BUSY THEN
		IF NOT fbAdsWrite.ERR THEN
			IF NOT bExecute THEN
				fbAdsWrite( WRITE := FALSE );
				nState	:= 0;
			ELSE
				nState	:= 20;
			END_IF
			bBusy	:= FALSE;
		ELSE
			bErr		:= TRUE;
			nErrId	:= fbAdsWrite.ERRID;
			nState	:= 20;
		END_IF
	END_IF
20:
	fbAdsWrite( WRITE := FALSE );
	bBusy	:= FALSE;
	IF NOT bExecute THEN
		nState	:= 0;
	END_IF
END_CASE
END_FUNCTION_BLOCK

(* POU ItpResetFastMFuncEx, ST *)
(*==========================================================*)
(* Name:			ItpResetFastMFuncEx   								*)
(* Desc:			resets specified fast m-func						*)
(* Author:	 	kbn														*)
(* Date:			26-September-2006										*)
(* last edit:	VER 6.2.33 						                  *)
(*==========================================================*)

